# B&R Automation Studio project NAINV104C00R8L515F00 (part 25)

#### Act_Background.st - Change By Project
```iecst
(** 2020-10-08 **)
ACTION Act_Background:

	//Resetting Physical Output
	memset(ADR(a_bPhysicalDO), 0, SIZEOF(a_bPhysicalDO));

	//Digital Output Mapping Physical Output With Config
	IF p_tyDOSettings.diSafetyRlyRst > 0 AND p_tyDOSettings.diSafetyRlyRst <= UDINT_TO_DINT(p_udiMax) THEN
		a_bPhysicalDO[p_tyDOSettings.diSafetyRlyRst]	:= p_bSafetyRlyRst;
	END_IF

	IF p_tyDOSettings.diTLRed > 0 AND p_tyDOSettings.diTLRed <= UDINT_TO_DINT(p_udiMax) THEN
		a_bPhysicalDO[p_tyDOSettings.diTLRed]			:= p_bTLRed;
	END_IF

	IF p_tyDOSettings.diTLAmber > 0 AND p_tyDOSettings.diTLAmber <= UDINT_TO_DINT(p_udiMax) THEN
		a_bPhysicalDO[p_tyDOSettings.diTLAmber]			:= p_bTLAmber;
	END_IF

	IF p_tyDOSettings.diTLGreen > 0 AND p_tyDOSettings.diTLGreen <= UDINT_TO_DINT(p_udiMax) THEN
		a_bPhysicalDO[p_tyDOSettings.diTLGreen]			:= p_bTLGreen;
	END_IF

	IF p_tyDOSettings.diTLWhite > 0 AND p_tyDOSettings.diTLWhite <= UDINT_TO_DINT(p_udiMax) THEN
		a_bPhysicalDO[p_tyDOSettings.diTLWhite]			:= p_bTLWhite;
	END_IF

	IF p_tyDOSettings.diTLBlue > 0 AND p_tyDOSettings.diTLBlue <= UDINT_TO_DINT(p_udiMax) THEN
		a_bPhysicalDO[p_tyDOSettings.diTLBlue]			:= p_bTLBlue;
	END_IF

	IF p_tyDOSettings.diBuz > 0 AND p_tyDOSettings.diBuz <= UDINT_TO_DINT(p_udiMax) THEN
		a_bPhysicalDO[p_tyDOSettings.diBuz]				:= p_bBuz;
	END_IF

	IF p_tyDOSettings.diDBA > 0 AND p_tyDOSettings.diDBA <= UDINT_TO_DINT(p_udiMax) THEN
		a_bPhysicalDO[p_tyDOSettings.diDBA]				:= p_bDBA;
	END_IF

	IF p_tyDOSettings.diDBAStat > 0 AND p_tyDOSettings.diDBAStat <= UDINT_TO_DINT(p_udiMax) THEN
		a_bPhysicalDO[p_tyDOSettings.diDBAStat]			:= p_bDBAStat;
	END_IF

	IF p_tyDOSettings.diUSB > 0 AND p_tyDOSettings.diUSB <= UDINT_TO_DINT(p_udiMax) THEN
		a_bPhysicalDO[p_tyDOSettings.diUSB]				:= p_bUSB;
	END_IF

	IF p_tyDOSettings.diUSB2 > 0 AND p_tyDOSettings.diUSB2 <= UDINT_TO_DINT(p_udiMax) THEN
		a_bPhysicalDO[p_tyDOSettings.diUSB2]			:= p_bUSB2;
	END_IF

	IF p_tyDOSettings.diConvMtrCW > 0 AND p_tyDOSettings.diConvMtrCW <= UDINT_TO_DINT(p_udiMax) THEN
		a_bPhysicalDO[p_tyDOSettings.diConvMtrCW]	:= p_bConvMtrCW;
	END_IF

	IF p_tyDOSettings.diConvMtrCCW > 0 AND p_tyDOSettings.diConvMtrCCW <= UDINT_TO_DINT(p_udiMax) THEN
		a_bPhysicalDO[p_tyDOSettings.diConvMtrCCW]	:= p_bConvMtrCCW;
	END_IF

	IF p_tyDOSettings.diStprUnblkCtrl > 0 AND p_tyDOSettings.diStprUnblkCtrl <= UDINT_TO_DINT(p_udiMax) THEN
		a_bPhysicalDO[p_tyDOSettings.diStprUnblkCtrl]	:= p_bStprUnblkCtrl;
	END_IF

	IF p_tyDOSettings.diStprBlkCtrl > 0 AND p_tyDOSettings.diStprBlkCtrl <= UDINT_TO_DINT(p_udiMax) THEN
		a_bPhysicalDO[p_tyDOSettings.diStprBlkCtrl]		:= p_bStprBlkCtrl;
	END_IF

	IF p_tyDOSettings.diInvertHome > 0 AND p_tyDOSettings.diInvertHome <= UDINT_TO_DINT(p_udiMax) THEN
		a_bPhysicalDO[p_tyDOSettings.diInvertHome]	:= p_bInvertHome;
	END_IF

	IF p_tyDOSettings.diInvertRemote > 0 AND p_tyDOSettings.diInvertRemote <= UDINT_TO_DINT(p_udiMax) THEN
		a_bPhysicalDO[p_tyDOSettings.diInvertRemote]	:= p_bInvertRemote;
	END_IF

	IF p_tyDOSettings.diInvertBrake > 0 AND p_tyDOSettings.diInvertBrake <= UDINT_TO_DINT(p_udiMax) THEN
		a_bPhysicalDO[p_tyDOSettings.diInvertBrake]	:= p_bInvertBrake;
	END_IF

	IF p_tyDOSettings.diClampControl > 0 AND p_tyDOSettings.diClampControl <= UDINT_TO_DINT(p_udiMax) THEN
		a_bPhysicalDO[p_tyDOSettings.diClampControl]	:= p_bClampControl;
	END_IF

	IF p_tyDOSettings.diUnclampControl > 0 AND p_tyDOSettings.diUnclampControl <= UDINT_TO_DINT(p_udiMax) THEN
		a_bPhysicalDO[p_tyDOSettings.diUnclampControl]	:= p_bUnclampControl;
	END_IF

	IF p_tyDOSettings.diMtrPwrRly > 0 AND p_tyDOSettings.diMtrPwrRly <= UDINT_TO_DINT(p_udiMax) THEN
		a_bPhysicalDO[p_tyDOSettings.diMtrPwrRly]	:= p_bMtrPwrRly;
	END_IF

	IF p_tyDOSettings.diInShutterOpenCtrl > 0 AND p_tyDOSettings.diInShutterOpenCtrl <= UDINT_TO_DINT(p_udiMax) THEN
		a_bPhysicalDO[p_tyDOSettings.diInShutterOpenCtrl]	:= p_bInShutterOpenCtrl;
	END_IF

	IF p_tyDOSettings.diInShutterCloseCtrl > 0 AND p_tyDOSettings.diInShutterCloseCtrl <= UDINT_TO_DINT(p_udiMax) THEN
		a_bPhysicalDO[p_tyDOSettings.diInShutterCloseCtrl]	:= p_bInShutterCloseCtrl;
	END_IF

	IF p_tyDOSettings.diOutShutterOpenCtrl > 0 AND p_tyDOSettings.diOutShutterOpenCtrl <= UDINT_TO_DINT(p_udiMax) THEN
		a_bPhysicalDO[p_tyDOSettings.diOutShutterOpenCtrl]	:= p_bOutShutterOpenCtrl;
	END_IF

	IF p_tyDOSettings.diOutShutterCloseCtrl > 0 AND p_tyDOSettings.diOutShutterCloseCtrl <= UDINT_TO_DINT(p_udiMax) THEN
		a_bPhysicalDO[p_tyDOSettings.diOutShutterCloseCtrl]	:= p_bOutShutterCloseCtrl;
	END_IF

	IF p_tyDOSettings.diClamp1Ctrl > 0 AND p_tyDOSettings.diClamp1Ctrl <= UDINT_TO_DINT(p_udiMax) THEN
		a_bPhysicalDO[p_tyDOSettings.diClamp1Ctrl]	:= p_bClamp1Ctrl;
	END_IF

	IF p_tyDOSettings.diUnClamp1Ctrl > 0 AND p_tyDOSettings.diUnClamp1Ctrl <= UDINT_TO_DINT(p_udiMax) THEN
		a_bPhysicalDO[p_tyDOSettings.diUnClamp1Ctrl]	:= p_bUnClamp1Ctrl;
	END_IF

	IF p_tyDOSettings.diClamp2Ctrl > 0 AND p_tyDOSettings.diClamp2Ctrl <= UDINT_TO_DINT(p_udiMax) THEN
		a_bPhysicalDO[p_tyDOSettings.diClamp2Ctrl]	:= p_bClamp2Ctrl;
	END_IF

	IF p_tyDOSettings.diUnClamp2Ctrl > 0 AND p_tyDOSettings.diUnClamp2Ctrl <= UDINT_TO_DINT(p_udiMax) THEN
		a_bPhysicalDO[p_tyDOSettings.diUnClamp2Ctrl]	:= p_bUnClamp2Ctrl;
	END_IF

	IF p_tyDOSettings.diClamp3Ctrl > 0 AND p_tyDOSettings.diClamp3Ctrl <= UDINT_TO_DINT(p_udiMax) THEN
		a_bPhysicalDO[p_tyDOSettings.diClamp3Ctrl]	:= p_bClamp3Ctrl; //
	END_IF

	IF p_tyDOSettings.diUnClamp3Ctrl > 0 AND p_tyDOSettings.diUnClamp3Ctrl <= UDINT_TO_DINT(p_udiMax) THEN
		a_bPhysicalDO[p_tyDOSettings.diUnClamp3Ctrl]	:= p_bUnClamp3Ctrl;
	END_IF

	// ADD
	IF p_bHermesUSCmdFeaturePause THEN
		IF p_tyHermesUSCmdPause.bFeatureRequestFrom  THEN
			//a_bPhysicalDO[p_tyDOSettings.diMachineSafetySigToUS]	:= p_tyHermesUSCmdPause.bMachineSafetySigTo;
			p_tyHermesUSCmdPause.bMachineSafetySigTo				:= p_bMachineSafetySigToUS;
		END_IF
		IF p_tyHermesUSCmdPause.bFeatureRequestTo THEN
			//a_bPhysicalDO[p_tyDOSettings.diTopCvrUnlckToUS]	:= p_tyHermesUSCmdPause.bUnlockCoverSigTo;
			p_tyHermesUSCmdPause.bUnlockCoverSigTo					:= p_bTopCvrUnlckToUS;
		END_IF
	ELSE
		IF p_tyDOSettings.diMachineSafetySigToUS > 0 AND p_tyDOSettings.diMachineSafetySigToUS  <= UDINT_TO_DINT(p_udiMax) THEN
			a_bPhysicalDO[p_tyDOSettings.diMachineSafetySigToUS]	:= p_bMachineSafetySigToUS;
		END_IF
		IF p_tyDOSettings.diTopCvrUnlckToUS > 0 AND p_tyDOSettings.diTopCvrUnlckToUS  <= UDINT_TO_DINT(p_udiMax) THEN
			a_bPhysicalDO[p_tyDOSettings.diTopCvrUnlckToUS]	:= p_bTopCvrUnlckToUS;
		END_IF
	END_IF
	IF p_bHermesDSCmdFeaturePause THEN
		IF p_tyHermesDSCmdPause.bFeatureRequestTo THEN
			//a_bPhysicalDO[p_tyDOSettings.diMachineSafetySigToDS]	:= p_tyHermesDSCmdPause.bMachineSafetySigTo;
			p_tyHermesDSCmdPause.bMachineSafetySigTo  				:= p_bMachineSafetySigToDS;
		END_IF
		IF p_tyHermesDSCmdPause.bFeatureRequestFrom THEN
			//a_bPhysicalDO[p_tyDOSettings.diTopCvrUnlckToDS]	:= p_tyHermesDSCmdPause.bUnlockCoverSigTo;
			p_tyHermesDSCmdPause.bUnlockCoverSigTo					:= p_bTopCvrUnlckToDS;
		END_IF
	ELSE
		IF p_tyDOSettings.diMachineSafetySigToDS  > 0 AND p_tyDOSettings.diMachineSafetySigToDS  <= UDINT_TO_DINT(p_udiMax) THEN
			a_bPhysicalDO[p_tyDOSettings.diMachineSafetySigToDS]	:= p_bMachineSafetySigToDS;
		END_IF
		IF p_tyDOSettings.diTopCvrUnlckToDS > 0 AND p_tyDOSettings.diTopCvrUnlckToDS  <= UDINT_TO_DINT(p_udiMax) THEN
			a_bPhysicalDO[p_tyDOSettings.diTopCvrUnlckToDS]	:= p_bTopCvrUnlckToDS;
		END_IF
	END_IF

	IF p_tyDOSettings.diSafetyTopCoverSWCoil1  > 0 AND p_tyDOSettings.diSafetyTopCoverSWCoil1  <= UDINT_TO_DINT(p_udiMax) THEN
		a_bPhysicalDO[p_tyDOSettings.diSafetyTopCoverSWCoil1]	:= p_bSafetyTopCoverSWCoil1;
	END_IF
	IF p_tyDOSettings.diCoverPBLED1 > 0 AND p_tyDOSettings.diCoverPBLED1  <= UDINT_TO_DINT(p_udiMax) THEN
		a_bPhysicalDO[p_tyDOSettings.diCoverPBLED1]	:= p_bCoverPBLED1;
	END_IF
	IF p_tyDOSettings.diBypassTopCover1 > 0 AND p_tyDOSettings.diBypassTopCover1  <= UDINT_TO_DINT(p_udiMax) THEN
		a_bPhysicalDO[p_tyDOSettings.diBypassTopCover1]	:= p_bBypsCoverSW1;
	END_IF

	//Update Output
	tyDOutput.bSafetyRlyRst			:= p_bSafetyRlyRst;
	tyDOutput.bTLWhite				:= p_bTLWhite;
	tyDOutput.bTLAmber				:= p_bTLAmber;
	tyDOutput.bTLGreen				:= p_bTLGreen;
	tyDOutput.bTLRed				:= p_bTLRed;
	tyDOutput.bTLBlue				:= p_bTLBlue;
	tyDOutput.bBuz					:= p_bBuz;
	tyDOutput.bUSB					:= p_bUSB;
	tyDOutput.bDBA					:= p_bDBA;
	tyDOutput.bDBAStat				:= p_bDBAStat;
	tyDOutput.bUSB2					:= p_bUSB2; //ADD_2023_0032B01
	tyDOutput.bConvMtrCW			:= p_bConvMtrCW;
	tyDOutput.bConvMtrCCW			:= p_bConvMtrCCW;
	tyDOutput.bStprUnblkCtrl		:= p_bStprUnblkCtrl;
	tyDOutput.bStprBlkCtrl			:= p_bStprBlkCtrl;
	tyDOutput.bInvertHome			:= p_bInvertHome;
	tyDOutput.bInvertRemote			:= p_bInvertRemote;
	tyDOutput.bInvertBrake			:= p_bInvertBrake;
	tyDOutput.bClampControl			:= p_bClampControl;
	tyDOutput.bUnclampControl		:= p_bUnclampControl;
	tyDOutput.bMtrPwrRly			:= p_bMtrPwrRly;
	tyDOutput.bInShutterOpenCtrl	:= p_bInShutterOpenCtrl;
	tyDOutput.bInShutterCloseCtrl	:= p_bInShutterCloseCtrl;
	tyDOutput.bOutShutterOpenCtrl	:= p_bOutShutterOpenCtrl;
	tyDOutput.bOutShutterCloseCtrl	:= p_bOutShutterCloseCtrl;
	tyDOutput.bClamp1Ctrl			:= p_bClamp1Ctrl;
	tyDOutput.bUnClamp1Ctrl			:= p_bUnClamp1Ctrl;
	tyDOutput.bClamp2Ctrl			:= p_bClamp2Ctrl;
	tyDOutput.bUnClamp2Ctrl			:= p_bUnClamp2Ctrl;
	tyDOutput.bClamp3Ctrl			:= p_bClamp3Ctrl;
	tyDOutput.bUnClamp3Ctrl			:= p_bUnClamp3Ctrl;

	// ADD
	tyDOutput.bMachineSafetySigToDS :=p_bMachineSafetySigToDS;
	tyDOutput.bMachineSafetySigToUS := p_bMachineSafetySigToUS;
	tyDOutput.bSafetyTopCoverSWCoil1 := p_bSafetyTopCoverSWCoil1;
	tyDOutput.bBypassTopCover1 := p_bBypsCoverSW1;
	tyDOutput.bCoverPBLED1 := p_bCoverPBLED1;
	tyDOutput.bTopCvrUnlckToDS := p_bMachineSafetySigToUS;
	tyDOutput.bTopCvrUnlckToUS := p_bMachineSafetySigToDS;
END_ACTION
```

#### InputRef.var - Change By Project
```iecst
(*2020-10-08*)
(**)
(*General*)
VAR
	p_eAct : REFERENCE TO eDOAction;
	p_udiMax : REFERENCE TO UDINT;
END_VAR
(**)
(*Configuration*)
VAR
	p_tyDOSettings : REFERENCE TO tyDigitalOutputSettings;
END_VAR
(**)
VAR
	p_bManual : REFERENCE TO BOOL;
	p_bSafetyRlyRst : REFERENCE TO BOOL;
	p_bTLRed : REFERENCE TO BOOL;
	p_bTLAmber : REFERENCE TO BOOL;
	p_bTLGreen : REFERENCE TO BOOL;
	p_bTLWhite : REFERENCE TO BOOL;
	p_bTLBlue : REFERENCE TO BOOL;
	p_bBuz : REFERENCE TO BOOL;
	p_bUSB : REFERENCE TO BOOL;
	p_bDBA : REFERENCE TO BOOL;
	p_bDBAStat : REFERENCE TO BOOL;
	p_bUSB2 : REFERENCE TO BOOL;
	p_bConvMtrCW : REFERENCE TO BOOL;
	p_bConvMtrCCW : REFERENCE TO BOOL;
	p_bStprUnblkCtrl : REFERENCE TO BOOL;
	p_bStprBlkCtrl : REFERENCE TO BOOL;
	p_bInvertBrake : REFERENCE TO BOOL;
	p_bInvertHome : REFERENCE TO BOOL;
	p_bInvertRemote : REFERENCE TO BOOL;
	p_bClampControl : REFERENCE TO BOOL;
	p_bUnclampControl : REFERENCE TO BOOL;
	p_bMtrPwrRly : REFERENCE TO BOOL;
	p_bInShutterOpenCtrl : REFERENCE TO BOOL;
	p_bInShutterCloseCtrl : REFERENCE TO BOOL;
	p_bOutShutterOpenCtrl : REFERENCE TO BOOL;
	p_bOutShutterCloseCtrl : REFERENCE TO BOOL;
	p_bClamp1Ctrl : REFERENCE TO BOOL;
	p_bUnClamp1Ctrl : REFERENCE TO BOOL;
	p_bClamp2Ctrl : REFERENCE TO BOOL;
	p_bUnClamp2Ctrl : REFERENCE TO BOOL;
	p_bClamp3Ctrl : REFERENCE TO BOOL;
	p_bUnClamp3Ctrl : REFERENCE TO BOOL;
END_VAR
(**)
VAR
	p_bLinkConvMtrSigOnOrLToR : REFERENCE TO BOOL;
	p_bLinkConvMtrDirOrRToL : REFERENCE TO BOOL;
	p_eLinkOpsInvertInvertCurrPos : REFERENCE TO eInvertPos;
	p_bLinkUIConvDCCtrl : REFERENCE TO BOOL;
	p_bLinkUIInvertDCCtrl : REFERENCE TO BOOL;
	p_usiLinkProdRcpCurrRcpMcMod : REFERENCE TO USINT;
	p_eConvStatus : REFERENCE TO eFBStatus;
	p_bLinkOpsInvertStepInitTwdStpr : REFERENCE TO BOOL;
	p_bLinkOpsInvertStepInitAwayStpr : REFERENCE TO BOOL;
END_VAR
(**)
VAR
	p_tyDI : REFERENCE TO tyDigitalInput;
END_VAR
(**)
VAR
	p_bBypsCoverSW1 : REFERENCE TO BOOL;
	p_bTopCvrUnlckToDS : REFERENCE TO BOOL;
	p_bTopCvrUnlckToUS : REFERENCE TO BOOL;
	p_bMachineSafetySigToDS : REFERENCE TO BOOL;
	p_bMachineSafetySigToUS : REFERENCE TO BOOL;
	p_bSafetyTopCoverSWCoil1 : REFERENCE TO BOOL;
	p_bCoverPBLED1 : REFERENCE TO BOOL;
END_VAR
(**)
VAR
	p_bHermesCmdInitialCompl : REFERENCE TO BOOL;
	p_bHermesUSCmdFeaturePause : REFERENCE TO BOOL;
	p_tyHermesUSCmdPause : REFERENCE TO tyHermesCommandPause;
	p_bHermesDSCmdFeaturePause : REFERENCE TO BOOL;
	p_tyHermesDSCmdPause : REFERENCE TO tyHermesCommandPause;
END_VAR
```

#### Local.var - Change By Project
```iecst
(*2020-10-08*)
(**)
(*Local Action, State & Status*)
VAR
	eAct : eDOAction := DOActIdle;
	eStat : eDOAction := DOActIdle;
	eStatus : eFBStatus := Idle;
	sStatTxt : STRING[200] := '';
	a_sStatText : ARRAY[0..50] OF STRING[200] := ['Idling','Resetting All Special Output','Turning On Bypass Cover Switch','Turning Off Bypass Cover Switch',47('')];
END_VAR
(**)
(*Local Alarm*)
(**)
(*Local Output*)
VAR
	tyDOutput : tyDigitalOutput;
END_VAR
(**)
(*Local Input*)
VAR
	tyDOSettings : tyDigitalOutputSettings;
END_VAR
(**)
VAR
	bManual : BOOL := FALSE;
	bSafetyRlyRst : BOOL := FALSE;
	bTLRed : BOOL := FALSE;
	bTLAmber : BOOL := FALSE;
	bTLGreen : BOOL := FALSE;
	bTLBlue : BOOL := FALSE;
	bTLWhite : BOOL := FALSE;
	bBuz : BOOL := FALSE;
	bUSB : BOOL := FALSE;
	bDBA : BOOL := FALSE;
	bDBAStat : BOOL := FALSE;
	bUSB2 : BOOL := FALSE;
	bConvMtrCW : BOOL := FALSE;
	bConvMtrCCW : BOOL := FALSE;
	bStprUnblkCtrl : BOOL := FALSE;
	bStprBlkCtrl : BOOL := FALSE;
	bInvertHome : BOOL := FALSE;
	bInvertRemote : BOOL := FALSE;
	bInvertBrake : BOOL := FALSE;
	bClampControl : BOOL := FALSE;
	bUnclampControl : BOOL := FALSE;
	bMtrPwrRly : BOOL := TRUE;
	bInShutterOpenCtrl : BOOL;
	bInShutterCloseCtrl : BOOL;
	bOutShutterOpenCtrl : BOOL;
	bOutShutterCloseCtrl : BOOL;
	bClamp1Ctrl : BOOL;
	bUnClamp1Ctrl : BOOL;
	bClamp2Ctrl : BOOL;
	bUnClamp2Ctrl : BOOL;
	bClamp3Ctrl : BOOL;
	bUnClamp3Ctrl : BOOL;
	bBypassTopCover1 : BOOL;
	bTopCvrUnlckToDS : BOOL;
	bTopCvrUnlckToUS : BOOL;
	bMachineSafetySigToDS : BOOL;
	bMachineSafetySigToUS : BOOL;
	bCoverPBLED1 : BOOL;
	bSafetyTopCoverSWCoil1 : BOOL;
END_VAR
(**)
(*Local*)
VAR
	bInitDone : BOOL;
	bInitialDone : BOOL;
	a_bPhysicalDO : ARRAY[1..c_udiDOutputMax] OF BOOL;
	eStatOld : eDOAction := DOActIdle;
	bHermesDummyMem : BOOL;
END_VAR
```

### Hermes.typ - Do Not Change!!!
```iecst
(*2019-05-04*)
(**)
(*Action*)

TYPE
	eHermesAction :
		(
		HermesActIdle,
		HermesActBGStartRun,
		HermesActBGStopRun,
		HermesActDeleteOldLog,
		HermesActCreateDir,
		HermesActWriteRetain,
		HermesActWriteRetainLane1,
		HermesActWriteRetainLane2,
		HermesActWriteRetainLane3,
		HermesActWriteRetainLane4,
		HermesActReadRetain,
		HermesActReadRetainLane1,
		HermesActReadRetainLane2,
		HermesActReadRetainLane3,
		HermesActReadRetainLane4,
		HermesActWriteConfig,
		HermesActReadConfig
		);
END_TYPE

(**)

TYPE
	tyHermesConfiguration : 	STRUCT
		a_tyUSParam : ARRAY[0..c_diHermesConfigMaxIdx]OF tyHermesUSParam;
		a_tyDSParam : ARRAY[0..c_diHermesConfigMaxIdx]OF tyHermesDSParam;
		tySvyParam : tyHermesSvyParam;
	END_STRUCT;
	tyHermesDSParam : 	STRUCT
		tSndAlive : TIME;
		tRcvAlive : TIME;
		sDownstreamInterfaceId : STRING[80]; (*The ID of the transportation interface on the downstream side*)
		uiSvrPort : UINT;
		iLaneID : INT;
		sMachineId : STRING[80] := '';
		sClientAddress : STRING[15] := '';
		uiClientPort : UINT;
		bFeatureCheckAliveResponse : BOOL;
		bFeatureBoardForecast : BOOL;
		bFeatureSendBoardInfo : BOOL;
		bFeatureCommand : BOOL;
	END_STRUCT;
	tyHermesUSParam : 	STRUCT
		tSndAlive : TIME;
		tRcvAlive : TIME;
		uiClntPort : UINT;
		iLaneID : INT;
		sMachineId : STRING[80] := '';
		sHostAddress : STRING[15] := '';
		uiHostPort : UINT;
		sUpstreamInterfaceId : STRING[80]; (*The ID of the transportation interface on the upstream side*)
		bFeatureCheckAliveResponse : BOOL;
		bFeatureBoardForecast : BOOL;
		bFeatureQueryBoardInfo : BOOL;
		bFeatureCommand : BOOL;
		bCmpTypeId : BOOL;
		bCmpParam : BOOL;
		bOverwrite : BOOL;
	END_STRUCT;
	tyHermesRmtParam : 	STRUCT
		uiSvrPort : UINT;
	END_STRUCT;
	tyHermesSvyParam : 	STRUCT
		tSndAlive : TIME;
		tRcvAlive : TIME;
		uiSvySvstemPort : UINT;
		iLaneID : INT;
		sMachineId : STRING[80];
		sClientAddress : STRING[15];
		uiClientPort : UINT;
		bFeatureCheckAliveResponse : BOOL;
		bFeatureConfiguration : BOOL;
		bFeatureBoardTracking : BOOL;
		bFeatureQueryWorkOrderInfo : BOOL;
		bFeatureSendWorkOrderInfo : BOOL;
		bFeatureInsertBrd : BOOL;
	END_STRUCT;
	tyHermesBrdAvlDat : 	STRUCT
		a_tyXMLTableDataBrdAvl : ARRAY[0..200]OF tyXMLTableDat;
		iXMLTableDataBrdAvlTtlIdx : INT;
		bNewBrdAvl : BOOL := TRUE;
	END_STRUCT;
END_TYPE
```

### Hermes.var - Change By Project
```iecst
(*2019-05-04*)
(**)
(*Action & State & Status*)
VAR
	p_HermesStat : UDINT;
	p_HermesStatus : UDINT;
	p_HermesStatTxt : UDINT;
END_VAR
(**)
(*Alarm*)
VAR
	p_HermesAlmData : UDINT;
END_VAR
(**)
(*Output*)
VAR
	p_HermesFileNotFound : UDINT;
	p_HermesConfiguration : UDINT;
	p_HermesConfigurationWr : UDINT;
	p_HermesUSParam1 : UDINT;
	p_HermesUSParam2 : UDINT;
	p_HermesUSParam3 : UDINT;
	p_HermesDSParam1 : UDINT;
	p_HermesDSParam2 : UDINT;
	p_HermesDSParam3 : UDINT;
	p_HermesSvyParam : UDINT;
	p_HermesBrdAvlDataTable1stZ : UDINT;
	p_HermesBrdAvlDataTtlIdx1stZ : UDINT;
	p_HermesBrdAvlDataNewBrdAvl1stZ : UDINT;
	p_HermesBrdAvlDataTableLastZ : UDINT;
	p_HermesBrdAvlDataTtlIdxLastZ : UDINT;
	p_HermesBrdAvlDataNewBrdAvlLastZ : UDINT;
	pa_HermesDSParam : UDINT;
	p_HermesReverseDS1SendBFId : UDINT;
	p_HermesReverseDS2SendBFId : UDINT;
	p_HermesSwitchtoReverseTransport : UDINT;
	p_HermesEntToReversePosition : UDINT;
	p_HermesCmdInitialCompl : UDINT;
	p_HermesUSCmdFeaturePause : UDINT;
	p_HermesUSCmdPause : UDINT;
	p_HermesDSCmdFeaturePause : UDINT;
	p_HermesDSCmdPause : UDINT;
END_VAR
```

### Program Logical/Hermes/Hermes (IEC, version 1.00.0) - 1.00.0 - NtHermes v5.00.0 , NtTCP v5.00.0 , NtMessage v5.00.0

#### Init.st - Change By Project
```iecst
(** 2019-05-04 **)
PROGRAM _INIT

	(* Always Change If Project Change *)

	//Pass Address To Global Address For External Use
	//Action, State & Status
	p_HermesStat	:= ADR(eStat);
	p_HermesStatus	:= ADR(eStatus);
	p_HermesStatTxt	:= ADR(sStatTxt);

	//Alarm
	p_HermesAlmData	:= ADR(tyAlmData);

	//Output
	p_HermesFileNotFound		:= ADR(bFileNotFound);
	p_HermesConfiguration		:= ADR(tyCurrConfiguration);
	p_HermesConfigurationWr	    := ADR(tyConfigurationWr);
	p_HermesUSParam1			:= ADR(tyCurrConfiguration.a_tyUSParam[0]);
	p_HermesUSParam2			:= ADR(tyCurrConfiguration.a_tyUSParam[1]);
	p_HermesUSParam3			:= ADR(tyCurrConfiguration.a_tyUSParam[2]);
	p_HermesDSParam1			:= ADR(tyCurrConfiguration.a_tyDSParam[0]);
	p_HermesDSParam2			:= ADR(tyCurrConfiguration.a_tyDSParam[1]);
	p_HermesDSParam3			:= ADR(tyCurrConfiguration.a_tyDSParam[2]);
	p_HermesSvyParam		    := ADR(tyCurrConfiguration.tySvyParam);
	p_HermesBrdAvlDataTable1stZ		    := ADR(a_tyHermesBrdAvlData[1].a_tyXMLTableDataBrdAvl); //Lane 1 First Zone Data, for B.F
	p_HermesBrdAvlDataTtlIdx1stZ    	:= ADR(a_tyHermesBrdAvlData[1].iXMLTableDataBrdAvlTtlIdx);  //Lane 1 First Zone Data, for B.F
	p_HermesBrdAvlDataNewBrdAvl1stZ	    := ADR(a_tyHermesBrdAvlData[1].bNewBrdAvl);  //Lane 1 First Zone Data, for B.F
	p_HermesBrdAvlDataTableLastZ		:= ADR(a_tyHermesBrdAvlData[1].a_tyXMLTableDataBrdAvl); //Lane 1 Last Zone Data,for B.A, adjust array no. accordingly
	p_HermesBrdAvlDataTtlIdxLastZ	    := ADR(a_tyHermesBrdAvlData[1].iXMLTableDataBrdAvlTtlIdx); //Lane 1 Last Zone Data,for B.A, adjust array no. accordingly
	p_HermesBrdAvlDataNewBrdAvlLastZ	:= ADR(a_tyHermesBrdAvlData[1].bNewBrdAvl); //Lane 1 Last Zone Data,for B.A, adjust array no. accordingly
	(* Always Change If Project Change *)
	p_HermesCmdInitialCompl		:= ADR(bCmdInitialCompl);

	//check route
	pa_HermesDSParam			:= ADR(tyCurrConfiguration.a_tyDSParam);

	//route output signal
	p_HermesReverseDS1SendBFId	:= ADR(usiReverseDS1SndBfWBrdID);
	p_HermesReverseDS2SendBFId	:= ADR(usiReverseDS2SndBfWBrdID);

	p_HermesSwitchtoReverseTransport := ADR(bSwitchtoReverseTransport);
	p_HermesEntToReversePosition := ADR(bEntToReversePosition);
	//p_HermesBrdAvlDataNewBrdAvlLastZ
END_PROGRAM
```

#### Act_InitGlobal.st - Change By Project
```iecst
(** 2019-05-04 **)
ACTION Act_InitGlobal:

	(* Always Change If Project Change *)

	//Pass Data To Link
	p_bLinkStartupRun ACCESS p_StartupRun;

	p_eLinkMcParamUSCommMod ACCESS p_McParamUSCommMod;
	p_eLinkMcParamUSComm2Mod ACCESS p_McParamUSComm2Mod;

	p_bLinkOpsInvertStepInitDone ACCESS p_OpsInvertStepInitDone;
	p_bLinkOpsInvertStepEntToEnd ACCESS p_OpsInvertStepEntToEnd;
	p_bLinkOpsInvertStepEntToInOff ACCESS p_OpsInvertStepEntToInOff;
	p_bLinkOpsInvertStepExitBrd ACCESS p_OpsInvertStepExitBrd;
	p_bLinkConvHvBrd ACCESS p_ConvHvBrd;//p_OpsInvertHvBrd;
	p_bLinkOpsInvertStepInvert ACCESS p_OpsInvertStepInvert;

	//p_tyUSHermestyBoardAvailable ACCESS p_USHermestyBoardAvailable;
	//Pass Data To Internal Use

	p_eAct ACCESS ADR(eAct);
	p_udiRstErr ACCESS p_RstErrReset;
	p_bPrep ACCESS p_NtParamHermesPrep;
	pa_tyUSParam ACCESS p_UIHermesUSParamWr;
	pa_tyDSParam ACCESS p_UIHermesDSParamWr;
	p_tySvyParam ACCESS p_UIHermesSvyParamWr; //HMI Svy Configure from UI
	p_tyRmtSetConfiguration ACCESS p_RmtHermesSetConfiguration; //US,DS SetConfigure from RmtHermes
	p_tySvySetConfiguration ACCESS p_SvyHermesSetConfiguration; //US,DS SetConfigure from SvyHermes

	//p_tySvySetConfiguration ACCESS p_SvyHermesSetConfiguration; //US,DS SetConfigure from SvyHermes
	p_bRmtPrep ACCESS p_NtParamHermesRmtPrep;
	p_bRmtEn ACCESS p_McParamHermesRmtEn;
	p_bSvyPrep ACCESS ADR(bSvyPrep);
	p_bSvyEn ACCESS ADR(bSvyEn);
	p_sRetainFileName1 ACCESS ADR(sRetainFileName1);
	p_sRetainFileName2 ACCESS ADR(sRetainFileName2);
	p_sRetainFileName3 ACCESS ADR(sRetainFileName3);
	p_sRetainFileName4 ACCESS ADR(sRetainFileName4);
	p_udiRetainDataAddr1 ACCESS ADR(udiRetainDataAddr1);
	p_udiRetainDataLen1 ACCESS ADR(udiRetainDataLen1);
	p_udiRetainDataAddr2 ACCESS ADR(udiRetainDataAddr2);
	p_udiRetainDataLen2 ACCESS ADR(udiRetainDataLen2);
	p_udiRetainDataAddr3 ACCESS ADR(udiRetainDataAddr3);
	p_udiRetainDataLen3 ACCESS ADR(udiRetainDataLen3);
	p_udiRetainDataAddr4 ACCESS ADR(udiRetainDataAddr4);
	p_udiRetainDataLen4 ACCESS ADR(udiRetainDataLen4);

	p_sConfigFileName ACCESS p_NtParamHermesConfigFileNm;
	p_sProgNm ACCESS p_NtParamHermesProgNm;
	p_bNtSettingsLoadDone ACCESS p_StartupNtSettingsLoadDone;
	p_bRmtHermesWriteConfig ACCESS p_RmtHermesWriteConfig;
	//p_bSvyHermesWriteConfig ACCESS p_SvyHermesWriteConfig;
	p_bUISaveHMIConfigure ACCESS p_UISaveHMIConfigure;
	p_bUISaveHMISvyConfig ACCESS p_UISaveHMISvyConfig;
	p_sMcId ACCESS p_McParamMcNm;

	p_bRmtFoundIndexUS1 ACCESS p_RmtHermesFoundIndexUS1;
	p_bRmtFoundIndexUS2 ACCESS p_RmtHermesFoundIndexUS2;
	p_bRmtFoundIndexUS3 ACCESS p_RmtHermesFoundIndexUS3;
	p_bRmtFoundIndexUS4 ACCESS p_RmtHermesFoundIndexUS4;
	p_bRmtFoundIndexDS1 ACCESS p_RmtHermesFoundIndexDS1;
	p_bRmtFoundIndexDS2 ACCESS p_RmtHermesFoundIndexDS2;
	p_bRmtFoundIndexDS3 ACCESS p_RmtHermesFoundIndexDS3;
	p_bRmtFoundIndexDS4 ACCESS p_RmtHermesFoundIndexDS4;
	p_udiRmtIndexUS1 ACCESS p_RmtHermesIndexUS1;
	p_udiRmtIndexUS2 ACCESS p_RmtHermesIndexUS2;
	p_udiRmtIndexUS3 ACCESS p_RmtHermesIndexUS3;
	p_udiRmtIndexUS4 ACCESS p_RmtHermesIndexUS4;
	p_udiRmtIndexDS1 ACCESS p_RmtHermesIndexDS1;
	p_udiRmtIndexDS2 ACCESS p_RmtHermesIndexDS2;
	p_udiRmtIndexDS3 ACCESS p_RmtHermesIndexDS3;
	p_udiRmtIndexDS4 ACCESS p_RmtHermesIndexDS4;

	p_bSvyFoundIndexUS1 ACCESS p_SvyHermesFoundIndexUS1;
	p_bSvyFoundIndexUS2 ACCESS p_SvyHermesFoundIndexUS2;
	p_bSvyFoundIndexUS3 ACCESS p_SvyHermesFoundIndexUS3;
	p_bSvyFoundIndexUS4 ACCESS p_SvyHermesFoundIndexUS4;
	p_bSvyFoundIndexDS1 ACCESS p_SvyHermesFoundIndexDS1;
	p_bSvyFoundIndexDS2 ACCESS p_SvyHermesFoundIndexDS2;
	p_bSvyFoundIndexDS3 ACCESS p_SvyHermesFoundIndexDS3;
	p_bSvyFoundIndexDS4 ACCESS p_SvyHermesFoundIndexDS4;
	p_udiSvyIndexUS1 ACCESS p_SvyHermesIndexUS1;
	p_udiSvyIndexUS2 ACCESS p_SvyHermesIndexUS2;
	p_udiSvyIndexUS3 ACCESS p_SvyHermesIndexUS3;
	p_udiSvyIndexUS4 ACCESS p_SvyHermesIndexUS4;
	p_udiSvyIndexDS1 ACCESS p_SvyHermesIndexDS1;
	p_udiSvyIndexDS2 ACCESS p_SvyHermesIndexDS2;
	p_udiSvyIndexDS3 ACCESS p_SvyHermesIndexDS3;
	p_udiSvyIndexDS4 ACCESS p_SvyHermesIndexDS4;

	//Command
	//Unlock Cover
	p_bNTParamUnlockCovPrep ACCESS p_NTParamUnlockCovPrep;
	p_bNTParamMachineSafetySig ACCESS p_NTParamMachineSafetySig;

	//route
	p_bOpsInvertStepInitDone ACCESS p_OpsInvertStepInitDone;
	p_bOpsInvertHvBrd ACCESS p_OpsInvertHvBrd;
	(* Always Change If Project Change *)

END_ACTION
```

#### InputRef_Link.var - Change By Project
```iecst
(*2019-05-04*)
(**)
VAR
	p_bLinkStartupRun : REFERENCE TO BOOL;
END_VAR
(**)
VAR
	p_eLinkMcParamUSCommMod : REFERENCE TO eMcSetCommMod;
	p_eLinkMcParamUSComm2Mod : REFERENCE TO eMcSetCommMod;
	pa_tyLinkXMLTableDataBrdAvl : REFERENCE TO ARRAY[0..200] OF tyXMLTableDat;
	p_iLinkXMLTableDataBrdAvlTtlIdx : REFERENCE TO INT;
END_VAR
(**)
VAR
	p_bLinkOpsInvertStepInitDone : REFERENCE TO BOOL;
	p_bLinkOpsInvertStepEntToEnd : REFERENCE TO BOOL;
	p_bLinkOpsInvertStepEntToInOff : REFERENCE TO BOOL;
	p_bLinkOpsInvertStepExitBrd : REFERENCE TO BOOL;
	p_bLinkConvHvBrd : REFERENCE TO BOOL;
	p_bLinkOpsInvertStepInvert : REFERENCE TO BOOL;
	p_tyUSHermestyBoardAvailable : REFERENCE TO tyHermesBoardAvailable;
END_VAR
(**)
VAR
	tyHermesBrdAvlData : tyHermesBrdAvlDat;
	a_tyHermesBrdAvlData : ARRAY[0..6] OF tyHermesBrdAvlDat; (*Cater Up to 6 Zones*)
	bHermesWriteRetain : BOOL;
	sLowerCase : STRING[254] := '';
END_VAR
```

#### Act_LinkAction.st - Change By Project
```iecst
(** 2019-05-04 **)
ACTION Act_LinkAction:

	IF p_bLinkStartupRun = TRUE THEN
		p_eAct ACCESS p_StartupHermesAct;
//	ELSIF p_bSvyHermesWriteConfig THEN
//		p_eAct ACCESS p_SvyHermesAct;
	ELSIF p_bRmtHermesWriteConfig THEN
		p_eAct ACCESS p_RmtHermesAct;
	ELSIF p_bUISaveHMIConfigure OR p_bUISaveHMISvyConfig THEN
		p_eAct ACCESS p_UIHermesAct;
	END_IF

END_ACTION
```

#### Act_LinkEn.st - Change By Project
```iecst
(** 2019-05-04 **)
ACTION Act_LinkEn:

	//Link bPrep, bEn & bDis

END_ACTION
```

#### Act_Link.st - Change By Project
```iecst
(** 2019-05-04 **)
ACTION Act_Link:

	IF p_bLinkStartupRun = FALSE THEN

		//Passing Board Available Memory
		//Init Board
		IF EDGEPOS(p_bLinkOpsInvertStepInitDone = TRUE) THEN

			IF p_bLinkConvHvBrd = FALSE THEN
				//tyHermesBrdAvlData.bNewBrdAvl	:= TRUE;
				a_tyHermesBrdAvlData[1].bNewBrdAvl := TRUE;
				bHermesWriteRetainLane1	:= TRUE;
			END_IF

		END_IF

		//Enter Board - US1
		IF EDGEPOS(p_bLinkConvHvBrd) AND (p_bLinkOpsInvertStepEntToEnd = TRUE OR p_bLinkOpsInvertStepEntToInOff) THEN

			IF p_eLinkMcParamUSCommMod = McSetCommModHermes THEN

				a_tyHermesBrdAvlData[1].a_tyXMLTableDataBrdAvl		:= pa_tyLinkXMLTableDataBrdAvl;
				a_tyHermesBrdAvlData[1].iXMLTableDataBrdAvlTtlIdx	:= p_iLinkXMLTableDataBrdAvlTtlIdx;
				a_tyHermesBrdAvlData[1].bNewBrdAvl					:= FALSE;

				bHermesWriteRetainLane1	:= TRUE;

			ELSE

				a_tyHermesBrdAvlData[1].bNewBrdAvl	:= TRUE;

				bHermesWriteRetainLane1	:= TRUE;

			END_IF

		END_IF

		//Exit Board
		IF p_bLinkOpsInvertStepExitBrd = TRUE AND EDGENEG(p_bLinkConvHvBrd) THEN
			a_tyHermesBrdAvlData[1].bNewBrdAvl	:= TRUE;

			bHermesWriteRetainLane1	:= TRUE;
		END_IF

		//Write Hermes Retain Data
		IF bHermesWriteRetainLane1 = TRUE AND eStatus <> Busy THEN
			p_eAct	:= HermesActWriteRetain;

			IF (eStat = HermesActWriteRetain) AND (eStatus = Done) THEN
				p_eAct				:= HermesActIdle;
				bHermesWriteRetainLane1	:= FALSE;
			END_IF
		END_IF

	END_IF

	IF EDGENEG(p_bLinkOpsInvertStepInvert) THEN
		FOR i := 0 TO 200 DO
			IF (a_tyHermesBrdAvlData[1].a_tyXMLTableDataBrdAvl[i].sTitle = 'AT') THEN
				fConvertToLower_254(ADR(sLowerCase) , a_tyHermesBrdAvlData[1].a_tyXMLTableDataBrdAvl[i].sValue);

				IF (sLowerCase = 'flippedboard') THEN
					IF a_tyHermesBrdAvlData[1].a_tyXMLTableDataBrdAvl[i+1].sTitle = 'AV' THEN
						IF p_tyUSHermestyBoardAvailable.tyData.eFlippedBoard = 1 THEN
							a_tyHermesBrdAvlData[1].a_tyXMLTableDataBrdAvl[i+1].sValue	:= '2';
						ELSIF  p_tyUSHermestyBoardAvailable.tyData.eFlippedBoard = 2 THEN
							a_tyHermesBrdAvlData[1].a_tyXMLTableDataBrdAvl[i+1].sValue	:= '1';
						ELSE
							a_tyHermesBrdAvlData[1].a_tyXMLTableDataBrdAvl[i+1].sValue	:= '0';
						END_IF

						EXIT;

					END_IF

				END_IF

			END_IF
		END_FOR
	END_IF

END_ACTION
```

#### Cyclic.st - Do Not Change!!!
```iecst
(** 2019-05-04 **)
PROGRAM _CYCLIC

	IF bInitDone = FALSE THEN
		bInitDone	:= TRUE;

		Act_InitLocal;
		Act_InitGlobal;

	ELSIF bInitialDone = FALSE THEN
		IF p_bNtSettingsLoadDone = TRUE THEN
			bInitialDone	:= TRUE;

			Act_Initial;
		END_IF

	ELSE

		Act_RstErr;
		Act_LinkAction;
		Act_Action;
		Act_LinkEn;

		IF (p_bPrep = TRUE) AND (p_bEn = TRUE) AND (p_bDis = FALSE) THEN
			Act_Background_Route;
			Act_Link;
			Act_Background;
			Act_Main;
			Act_Background_Command;

		ELSE
			IF eStat <> HermesActIdle THEN
				eStatus	:= Done;
			ELSE
				eStatus	:= Idle;
			END_IF
		END_IF

		Act_Alarm;

	END_IF

END_PROGRAM
```

#### Act_RstErr.st - Do Not Change!!!
```iecst
(** 2019-05-04 **)
ACTION Act_RstErr:

	IF p_udiRstErr <> udiRstErrOld THEN
		bRstErr			:= TRUE;
		udiRstErrOld	:= p_udiRstErr;
	ELSE
		bRstErr			:= FALSE;
	END_IF

END_ACTION
```

#### Act_InitLocal.st - Do Not Change!!!
```iecst
(** 2019-05-04 **)
ACTION Act_InitLocal:

	//Input Reference Link To Local Variable
	p_eAct ACCESS ADR(eAct);
	p_udiRstErr ACCESS ADR(udiRstErr);
	p_bPrep ACCESS ADR(bPrep);
	p_bEn ACCESS ADR(bEn);
	p_bDis ACCESS ADR(bDis);
	pa_tyUSParam ACCESS ADR(a_tyUSParam);
	pa_tyDSParam ACCESS ADR(a_tyDSParam);
	p_tyRmtParam ACCESS ADR(tyRmtParam);
	p_tySvyParam ACCESS ADR(tySvyParam);
	p_tyRmtSetConfiguration ACCESS ADR(tyRmtSetConfiguration);
	p_tySvySetConfiguration ACCESS ADR(tySvySetConfiguration);

	p_bRmtPrep ACCESS ADR(bRmtPrep);
	p_bRmtEn ACCESS ADR(bRmtEn);
	p_bSvyPrep ACCESS ADR(bSvyPrep);
	p_bSvyEn ACCESS ADR(bSvyEn);
	p_sRetainFileName1 ACCESS ADR(sRetainFileName1);
	p_sRetainFileName2 ACCESS ADR(sRetainFileName2);
	p_sRetainFileName3 ACCESS ADR(sRetainFileName3);
	p_sRetainFileName4 ACCESS ADR(sRetainFileName4);
	p_udiRetainDataAddr1 ACCESS ADR(udiRetainDataAddr1);
	p_udiRetainDataLen1 ACCESS ADR(udiRetainDataLen1);
	p_udiRetainDataAddr2 ACCESS ADR(udiRetainDataAddr2);
	p_udiRetainDataLen2 ACCESS ADR(udiRetainDataLen2);
	p_udiRetainDataAddr3 ACCESS ADR(udiRetainDataAddr3);
	p_udiRetainDataLen3 ACCESS ADR(udiRetainDataLen3);
	p_udiRetainDataAddr4 ACCESS ADR(udiRetainDataAddr4);
	p_udiRetainDataLen4 ACCESS ADR(udiRetainDataLen4);

	p_sConfigFileName ACCESS ADR(sConfigFileName);
	p_sProgNm ACCESS ADR(sProgNm);
	p_bNtSettingsLoadDone ACCESS ADR(bNtSettingsLoadDone);
	p_bRmtHermesWriteConfig ACCESS ADR(bRmtHermesWriteConfig);
	p_bSvyHermesWriteConfig ACCESS ADR(bSvyHermesWriteConfig);
	p_bUISaveHMIConfigure ACCESS ADR(bUISaveHMIConfigure);
	p_bUISaveHMISvyConfig ACCESS ADR(bUISaveHMISvyConfig);
	p_sMcId ACCESS ADR(sMcId);

	p_bRmtFoundIndexUS1 ACCESS ADR(bRmtFoundIndexUS1);
	p_bRmtFoundIndexUS2 ACCESS ADR(bRmtFoundIndexUS2);
	p_bRmtFoundIndexUS3 ACCESS ADR(bRmtFoundIndexUS3);
	p_bRmtFoundIndexUS4 ACCESS ADR(bRmtFoundIndexUS4);
	p_bRmtFoundIndexDS1 ACCESS ADR(bRmtFoundIndexDS1);
	p_bRmtFoundIndexDS2 ACCESS ADR(bRmtFoundIndexDS2);
	p_bRmtFoundIndexDS3 ACCESS ADR(bRmtFoundIndexDS3);
	p_bRmtFoundIndexDS4 ACCESS ADR(bRmtFoundIndexDS4);
	p_udiRmtIndexUS1 ACCESS ADR(udiRmtIndexUS1);
	p_udiRmtIndexUS2 ACCESS ADR(udiRmtIndexUS2);
	p_udiRmtIndexUS3 ACCESS ADR(udiRmtIndexUS3);
	p_udiRmtIndexUS4 ACCESS ADR(udiRmtIndexUS4);
	p_udiRmtIndexDS1 ACCESS ADR(udiRmtIndexDS1);
	p_udiRmtIndexDS2 ACCESS ADR(udiRmtIndexDS2);
	p_udiRmtIndexDS3 ACCESS ADR(udiRmtIndexDS3);
	p_udiRmtIndexDS4 ACCESS ADR(udiRmtIndexDS4);

	p_bSvyFoundIndexUS1 ACCESS ADR(bSvyFoundIndexUS1);
	p_bSvyFoundIndexUS2 ACCESS ADR(bSvyFoundIndexUS2);
	p_bSvyFoundIndexUS3 ACCESS ADR(bSvyFoundIndexUS3);
	p_bSvyFoundIndexUS4 ACCESS ADR(bSvyFoundIndexUS4);
	p_bSvyFoundIndexDS1 ACCESS ADR(bSvyFoundIndexDS1);
	p_bSvyFoundIndexDS2 ACCESS ADR(bSvyFoundIndexDS2);
	p_bSvyFoundIndexDS3 ACCESS ADR(bSvyFoundIndexDS3);
	p_bSvyFoundIndexDS4 ACCESS ADR(bSvyFoundIndexDS4);

	p_udiSvyIndexUS1 ACCESS ADR(udiSvyIndexUS1);
	p_udiSvyIndexUS2 ACCESS ADR(udiSvyIndexUS2);
	p_udiSvyIndexUS3 ACCESS ADR(udiSvyIndexUS3);
	p_udiSvyIndexUS4 ACCESS ADR(udiSvyIndexUS4);
	p_udiSvyIndexDS1 ACCESS ADR(udiSvyIndexDS1);
	p_udiSvyIndexDS2 ACCESS ADR(udiSvyIndexDS2);
	p_udiSvyIndexDS3 ACCESS ADR(udiSvyIndexDS3);
	p_udiSvyIndexDS4 ACCESS ADR(udiSvyIndexDS4);

	p_bReverseReceiveRoute ACCESS ADR(bReverseReceiveRoute);
	p_bReverseSentRoute ACCESS ADR(bReverseSendRoute);

	p_bManualRmvRoute ACCESS ADR(bManualRmvRoute);
	p_bReturnRoute ACCESS ADR(bReturnRoute);
	p_bNomRouteEn ACCESS ADR(bNomRouteEn);
END_ACTION
```

#### Act_Initial.st - Do Not Change!!!
```iecst
(** 2019-05-04 **)
ACTION Act_Initial:
	//Initial

	//Retain Data
	p_udiRetainDataAddr1	:= ADR(a_tyHermesBrdAvlData);
	p_udiRetainDataLen1	:= SIZEOF(a_tyHermesBrdAvlData);

	sStatTxt	:= a_sStatText[eStat];

	fbDirCreate1.sDevice	:= 'F';
	fbDirCreate1.sDirName	:= 'User';
	fbDirCreate1(bEn := FALSE);

	fbDirCreate2.sDevice	:= 'User';
	fbDirCreate2.sDirName	:= 'Retain';
	fbDirCreate2(bEn := FALSE);

	fbDirCreate3.sDevice	:= 'User';
	fbDirCreate3.sDirName	:= 'Log';
	fbDirCreate3(bEn := FALSE);

	fbDirCreate4.sDevice	:= 'User';
	fbDirCreate4.sDirName	:= 'MachineParameter';
	fbDirCreate4(bEn := FALSE);

	fbFileRead1.sDevice			:= 'McParam';
	fbFileRead1.sFile			:= p_sConfigFileName;
	fbFileRead1.udiOffset		:= 0;
	fbFileRead1.p_Dest			:= ADR(tyCurrConfiguration);
	fbFileRead1.udiLen			:= SIZEOF(tyCurrConfiguration);
	fbFileRead1(bEn := FALSE);

	fbFileWrite1.sDevice		:= 'McParam';
	fbFileWrite1.sFile			:= p_sConfigFileName;
	fbFileWrite1.udiOffset		:= 0;
	fbFileWrite1.p_Src			:= ADR(tyConfigurationWr);
	fbFileWrite1.udiLen			:= SIZEOF(tyConfigurationWr);
	fbFileWrite1.udiOption		:= 0;
	fbFileWrite1(bEn := FALSE);

	fbFileRead2.sDevice			:= 'Retain';
	fbFileRead2.sFile			:= p_sRetainFileName1;
	fbFileRead2.udiOffset		:= 0;
	fbFileRead2.p_Dest			:= p_udiRetainDataAddr1;
	fbFileRead2.udiLen			:= p_udiRetainDataLen1;
	fbFileRead2(bEn := FALSE);

	fbFileWrite2.sDevice		:= 'Retain';
	fbFileWrite2.sFile			:= p_sRetainFileName1;
	fbFileWrite2.udiOffset		:= 0;
	fbFileWrite2.p_Src			:= p_udiRetainDataAddr1;
	fbFileWrite2.udiLen			:= p_udiRetainDataLen1;
	fbFileWrite2.udiOption		:= 0;
	fbFileWrite2(bEn := FALSE);

	fbFileRead3.sDevice			:= 'Retain';
	fbFileRead3.sFile			:= p_sRetainFileName2;
	fbFileRead3.udiOffset		:= 0;
	fbFileRead3.p_Dest			:= p_udiRetainDataAddr2;
	fbFileRead3.udiLen			:= p_udiRetainDataLen2;
	fbFileRead3(bEn := FALSE);

	fbFileWrite3.sDevice		:= 'Retain';
	fbFileWrite3.sFile			:= p_sRetainFileName2;
	fbFileWrite3.udiOffset		:= 0;
	fbFileWrite3.udiOption		:= 0;
	fbFileWrite3.p_Src			:= p_udiRetainDataAddr2;
	fbFileWrite3.udiLen			:= p_udiRetainDataLen2;
	fbFileWrite3(bEn := FALSE);

	fbFileRead4.sDevice			:= 'Retain';
	fbFileRead4.sFile			:= p_sRetainFileName3;
	fbFileRead4.udiOffset		:= 0;
	fbFileRead4.p_Dest			:= p_udiRetainDataAddr3;
	fbFileRead4.udiLen			:= p_udiRetainDataLen3;
	fbFileRead4(bEn := FALSE);

	fbFileWrite4.sDevice		:= 'Retain';
	fbFileWrite4.sFile			:= p_sRetainFileName3;
	fbFileWrite4.udiOffset		:= 0;
	fbFileWrite4.udiOption		:= 0;
	fbFileWrite4.p_Src			:= p_udiRetainDataAddr3;
	fbFileWrite4.udiLen			:= p_udiRetainDataLen3;
	fbFileWrite4(bEn := FALSE);

	fbFileRead5.sDevice			:= 'Retain';
	fbFileRead5.sFile			:= p_sRetainFileName4;
	fbFileRead5.udiOffset		:= 0;
	fbFileRead5.p_Dest			:= p_udiRetainDataAddr4;
	fbFileRead5.udiLen			:= p_udiRetainDataLen4;
	fbFileRead5(bEn := FALSE);

	fbFileWrite5.sDevice		:= 'Retain';
	fbFileWrite5.sFile			:= p_sRetainFileName4;
	fbFileWrite5.udiOffset		:= 0;
	fbFileWrite5.udiOption		:= 0;
	fbFileWrite5.p_Src			:= p_udiRetainDataAddr4;
	fbFileWrite5.udiLen			:= p_udiRetainDataLen4;
	fbFileWrite5(bEn := FALSE);

	//Command
	memset(ADR(a_tyCommandProcessList),0,SIZEOF(a_tyCommandProcessList));
	usiProcessCmdBffr := 0;
	usiUSIdent  := fHermesAddOneCommandGate(TRUE,p_USHermesCommandParam,ADR(tyCurrConfiguration.a_tyUSParam[0].sUpstreamInterfaceId),p_McParamUSCommMod,ADR(a_tyCommandProcessList),ADR(usiProcessCmdBffr));
	usiDSIdent  := fHermesAddOneCommandGate(FALSE,p_DSHermesCommandParam,ADR(tyCurrConfiguration.a_tyDSParam[0].sDownstreamInterfaceId),p_McParamDSCommMod,ADR(a_tyCommandProcessList),ADR(usiProcessCmdBffr));
	usiUSIdent2 := fHermesAddOneCommandGate(TRUE,p_USHermes2CommandParam,ADR(tyCurrConfiguration.a_tyUSParam[1].sUpstreamInterfaceId),p_McParamUSComm2Mod,ADR(a_tyCommandProcessList),ADR(usiProcessCmdBffr));

	//output
	bCmdInitialCompl := TRUE;

	//tyCurrConfiguration
	//Feature(Machine Safety)
	p_HermesUSCmdFeaturePause := ADR(tyCurrConfiguration.a_tyUSParam[0].bFeatureCommand);
	p_HermesUSCmdPause := ADR(a_tyCommandPause[usiUSIdent]);
	p_HermesDSCmdFeaturePause := ADR(tyCurrConfiguration.a_tyDSParam[0].bFeatureCommand);
	p_HermesDSCmdPause := ADR(a_tyCommandPause[usiDSIdent]);
	a_tyCommandPause[usiUSIdent].bFeatureRequestFrom :=  p_bNTParamMachineSafetySig;
	a_tyCommandPause[usiUSIdent].bFeatureRequestTo   :=  p_bNTParamUnlockCovPrep;

	a_tyCommandPause[usiDSIdent].bFeatureRequestFrom := p_bNTParamMachineSafetySig;
	a_tyCommandPause[usiDSIdent].bFeatureRequestTo	:=  p_bNTParamUnlockCovPrep;

	//Feature(Oven Info)
	//p_HermesUSCmdFeaturePause := ADR(tyCurrConfiguration.a_tyUSParam[1].bFeatureCommand);
	//p_HermesUSCmdPause := ADR(a_tyCommandPause[usiUSIdent2]);
	//a_tyCommandLockInputConv[usiUSIdent].bFeatureLockConvTo   :=  p_bNTParamOvenInfoAPrep;
	//a_tyCommandLockInputConv[usiDSIdent].bFeatureLockConvFrom := p_bNTParamOvenInfoAPrep;
	//a_tyCommandLockInputConv[usiUSIdent2].bFeatureLockConvTo  :=  p_bNTParamOvenInfoBPrep;

END_ACTION
```

#### Act_Main.st - Do Not Change!!!
```iecst
(** 2021-08-01 **)
ACTION Act_Main:

	IF eStatOld <> eStat THEN
		fbDirCreate1(bEn := FALSE);
		fbDirCreate2(bEn := FALSE);
		fbDirCreate3(bEn := FALSE);
		fbDirCreate4(bEn := FALSE);
		fbFileRead1(bEn := FALSE);
		fbFileWrite1(bEn := FALSE);
		fbFileRead2(bEn := FALSE);
		fbFileWrite2(bEn := FALSE);
		fbFileRead3(bEn := FALSE);
		fbFileWrite3(bEn := FALSE);
		fbFileRead4(bEn := FALSE);
		fbFileWrite4(bEn := FALSE);
		fbFileRead5(bEn := FALSE);
		fbFileWrite5(bEn := FALSE);
		usiStep			:= 0;
		bFileNotFound	:= FALSE;

		sStatTxt	:= a_sStatText[eStat];

		eStatOld	:= eStat;

		eStatus		:= Busy;
	END_IF

	//Main
	CASE eStat OF

		HermesActIdle:
			eStatus	:= Idle;

		HermesActCreateDir:
			IF eStatus = Idle OR eStatus = Busy THEN

				eStatus	:= Busy;

				CASE usiStep OF
					0:
						fbDirCreate1(bEn := TRUE);
						IF fbDirCreate1.udiStatus = 0 THEN
							usiStep	:= 1;
						ELSIF fbDirCreate1.udiStatus < 65534 THEN
							eStatus		:= Error;

							IF fbDirCreate1.udiStatus = 1908 THEN
								udiStatus	:= 10000;	//Create User Directory Error
							ELSE
								udiStatus	:= fbDirCreate1.udiStatus;
							END_IF
						END_IF

					1:
						fbDirCreate2(bEn := TRUE);
						IF fbDirCreate2.udiStatus = 0 THEN
							usiStep	:= 2;
						ELSIF fbDirCreate2.udiStatus < 65534 THEN
							eStatus		:= Error;

							IF fbDirCreate2.udiStatus = 1908 THEN
								udiStatus	:= 10001;	//Create Retain Directory Error
							ELSE
								udiStatus	:= fbDirCreate2.udiStatus;
							END_IF
						END_IF

					2:
						fbDirCreate3(bEn := TRUE);
						IF fbDirCreate3.udiStatus = 0 THEN
							usiStep	:= 3;
						ELSIF fbDirCreate3.udiStatus < 65534 THEN
							eStatus		:= Error;

							IF fbDirCreate3.udiStatus = 1908 THEN
								udiStatus	:= 10010;	//Create Log Directory Error
							ELSE
								udiStatus	:= fbDirCreate3.udiStatus;
							END_IF
						END_IF

					3:
						fbDirCreate4(bEn := TRUE);
						IF fbDirCreate4.udiStatus = 0 THEN
							eStatus	:= Done;
						ELSIF fbDirCreate4.udiStatus < 65534 THEN
							eStatus		:= Error;

							IF fbDirCreate4.udiStatus = 1908 THEN
								udiStatus	:= 10011;	//Create Machine Parameter Directory Error
							ELSE
								udiStatus	:= fbDirCreate4.udiStatus;
							END_IF
						END_IF

				END_CASE

			END_IF

		HermesActReadRetainLane1:
			IF eStatus = Idle OR eStatus = Busy THEN

				eStatus	:= Busy;

				fbFileRead2(bEn := TRUE);

				IF fbFileRead2.udiStatus = 0 THEN
					eStatus	:= Done;
				ELSIF fbFileRead2.udiStatus < 65534 THEN
					eStatus	:= Error;

					IF fbFileRead2.udiStatus = 1900 THEN
						udiStatus	:= 10002;	//File Open Error While Reading Retain File
					ELSIF fbFileRead2.udiStatus = 1902 THEN
						udiStatus	:= 10003;	//File Read Error While Reading Retain File
					ELSIF fbFileRead2.udiStatus = 1904 THEN
						udiStatus	:= 10004;	//File Close Error While Reading Retain File
					ELSIF fbFileRead2.udiStatus = 1915 THEN
						eStatus			:= Done;
						bFileNotFound	:= TRUE;
					ELSE
						udiStatus	:= fbFileRead2.udiStatus;
					END_IF
				END_IF

			END_IF

		HermesActWriteRetainLane1:
			IF eStatus = Idle OR eStatus = Busy THEN

				eStatus	:= Busy;

				fbFileWrite2(bEn := TRUE);

				IF fbFileWrite2.udiStatus = 0 THEN
					eStatus	:= Done;
				ELSIF fbFileWrite2.udiStatus < 65534 THEN
					eStatus	:= Error;

					IF fbFileWrite2.udiStatus = 1900 THEN
						udiStatus	:= 10005;	//File Open Error While Writing Retain File
					ELSIF fbFileWrite2.udiStatus = 1901 THEN
						udiStatus	:= 10006;	//File Create Error While Writing Retain File
					ELSIF fbFileWrite2.udiStatus = 1903 THEN
						udiStatus	:= 10007;	//File Write Error While Writing Retain File
					ELSIF fbFileWrite2.udiStatus = 1904 THEN
						udiStatus	:= 10008;	//File Close Error While Writing Retain File
					ELSIF fbFileWrite2.udiStatus = 1914 THEN
						udiStatus	:= 10009;	//Directory Does Not Exist While Writing Retain File
					ELSE
						udiStatus	:= fbFileWrite2.udiStatus;
					END_IF
				END_IF

			END_IF

		HermesActReadRetainLane2:
			IF eStatus = Idle OR eStatus = Busy THEN

				eStatus	:= Busy;

				fbFileRead3(bEn := TRUE);

				IF fbFileRead3.udiStatus = 0 THEN
					eStatus	:= Done;
				ELSIF fbFileRead3.udiStatus < 65534 THEN
					eStatus	:= Error;

					IF fbFileRead3.udiStatus = 1900 THEN
						udiStatus	:= 10032;	//File Open Error While Reading Retain File
					ELSIF fbFileRead3.udiStatus = 1902 THEN
						udiStatus	:= 10033;	//File Read Error While Reading Retain File
					ELSIF fbFileRead3.udiStatus = 1904 THEN
						udiStatus	:= 10034;	//File Close Error While Reading Retain File
					ELSIF fbFileRead3.udiStatus = 1915 THEN
						eStatus			:= Done;
						bFileNotFound	:= TRUE;
					ELSE
						udiStatus	:= fbFileRead3.udiStatus;
					END_IF
				END_IF

			END_IF

		HermesActWriteRetainLane2:
			IF eStatus = Idle OR eStatus = Busy THEN

				eStatus	:= Busy;

				fbFileWrite3(bEn := TRUE);

				IF fbFileWrite3.udiStatus = 0 THEN
					eStatus	:= Done;
				ELSIF fbFileWrite3.udiStatus < 65534 THEN
					eStatus	:= Error;

					IF fbFileWrite3.udiStatus = 1900 THEN
						udiStatus	:= 10035;	//File Open Error While Writing Retain File
					ELSIF fbFileWrite3.udiStatus = 1901 THEN
						udiStatus	:= 10036;	//File Create Error While Writing Retain File
					ELSIF fbFileWrite3.udiStatus = 1903 THEN
						udiStatus	:= 10037;	//File Write Error While Writing Retain File
					ELSIF fbFileWrite3.udiStatus = 1904 THEN
						udiStatus	:= 10038;	//File Close Error While Writing Retain File
					ELSIF fbFileWrite3.udiStatus = 1914 THEN
						udiStatus	:= 10039;	//Directory Does Not Exist While Writing Retain File
					ELSE
						udiStatus	:= fbFileWrite3.udiStatus;
					END_IF
				END_IF

			END_IF

		HermesActReadRetainLane3:
			IF eStatus = Idle OR eStatus = Busy THEN

				eStatus	:= Busy;

				fbFileRead4(bEn := TRUE);

				IF fbFileRead4.udiStatus = 0 THEN
					eStatus	:= Done;
				ELSIF fbFileRead4.udiStatus < 65534 THEN
					eStatus	:= Error;

					IF fbFileRead4.udiStatus = 1900 THEN
						udiStatus	:= 10042;	//File Open Error While Reading Retain File
					ELSIF fbFileRead4.udiStatus = 1902 THEN
						udiStatus	:= 10043;	//File Read Error While Reading Retain File
					ELSIF fbFileRead4.udiStatus = 1904 THEN
						udiStatus	:= 10044;	//File Close Error While Reading Retain File
					ELSIF fbFileRead4.udiStatus = 1915 THEN
						eStatus			:= Done;
						bFileNotFound	:= TRUE;
					ELSE
						udiStatus	:= fbFileRead4.udiStatus;
					END_IF
				END_IF

			END_IF

		HermesActWriteRetainLane3:
			IF eStatus = Idle OR eStatus = Busy THEN

				eStatus	:= Busy;

				fbFileWrite4(bEn := TRUE);

				IF fbFileWrite4.udiStatus = 0 THEN
					eStatus	:= Done;
				ELSIF fbFileWrite4.udiStatus < 65534 THEN
					eStatus	:= Error;

					IF fbFileWrite4.udiStatus = 1900 THEN
						udiStatus	:= 10045;	//File Open Error While Writing Retain File
					ELSIF fbFileWrite4.udiStatus = 1901 THEN
						udiStatus	:= 10046;	//File Create Error While Writing Retain File
					ELSIF fbFileWrite4.udiStatus = 1903 THEN
						udiStatus	:= 10047;	//File Write Error While Writing Retain File
					ELSIF fbFileWrite4.udiStatus = 1904 THEN
						udiStatus	:= 10048;	//File Close Error While Writing Retain File
					ELSIF fbFileWrite4.udiStatus = 1914 THEN
						udiStatus	:= 10049;	//Directory Does Not Exist While Writing Retain File
					ELSE
						udiStatus	:= fbFileWrite4.udiStatus;
					END_IF
				END_IF

			END_IF

		HermesActReadRetainLane4:
			IF eStatus = Idle OR eStatus = Busy THEN

				eStatus	:= Busy;

				fbFileRead5(bEn := TRUE);

				IF fbFileRead5.udiStatus = 0 THEN
					eStatus	:= Done;
				ELSIF fbFileRead5.udiStatus < 65534 THEN
					eStatus	:= Error;

					IF fbFileRead5.udiStatus = 1900 THEN
						udiStatus	:= 10052;	//File Open Error While Reading Retain File
					ELSIF fbFileRead5.udiStatus = 1902 THEN
						udiStatus	:= 10053;	//File Read Error While Reading Retain File
					ELSIF fbFileRead5.udiStatus = 1904 THEN
						udiStatus	:= 10054;	//File Close Error While Reading Retain File
					ELSIF fbFileRead5.udiStatus = 1915 THEN
						eStatus			:= Done;
						bFileNotFound	:= TRUE;
					ELSE
						udiStatus	:= fbFileRead5.udiStatus;
					END_IF
				END_IF

			END_IF

		HermesActWriteRetainLane4:
			IF eStatus = Idle OR eStatus = Busy THEN

				eStatus	:= Busy;

				fbFileWrite5(bEn := TRUE);

				IF fbFileWrite5.udiStatus = 0 THEN
					eStatus	:= Done;
				ELSIF fbFileWrite5.udiStatus < 65534 THEN
					eStatus	:= Error;

					IF fbFileWrite5.udiStatus = 1900 THEN
						udiStatus	:= 10055;	//File Open Error While Writing Retain File
					ELSIF fbFileWrite5.udiStatus = 1901 THEN
						udiStatus	:= 10056;	//File Create Error While Writing Retain File
					ELSIF fbFileWrite5.udiStatus = 1903 THEN
						udiStatus	:= 10057;	//File Write Error While Writing Retain File
					ELSIF fbFileWrite5.udiStatus = 1904 THEN
						udiStatus	:= 10058;	//File Close Error While Writing Retain File
					ELSIF fbFileWrite5.udiStatus = 1914 THEN
						udiStatus	:= 10059;	//Directory Does Not Exist While Writing Retain File
					ELSE
						udiStatus	:= fbFileWrite5.udiStatus;
					END_IF
				END_IF

			END_IF

		HermesActReadConfig:
			IF eStatus = Idle OR eStatus = Busy THEN

				eStatus	:= Busy;

				fbFileRead1(bEn := TRUE);

				IF fbFileRead1.udiStatus = 0 THEN
					eStatus	:= Done;
					tyConfigurationWr := tyCurrConfiguration;
				ELSIF fbFileRead1.udiStatus < 65534 THEN
					eStatus	:= Error;

					IF fbFileRead1.udiStatus = 1900 THEN
						udiStatus	:= 10012;	//File Open Error While Reading Config File
					ELSIF fbFileRead1.udiStatus = 1902 THEN
						udiStatus	:= 10013;	//File Read Error While Reading Config File
					ELSIF fbFileRead1.udiStatus = 1904 THEN
						udiStatus	:= 10014;	//File Close Error While Reading Config File
					ELSIF fbFileRead1.udiStatus = 1915 THEN
						eStatus			:= Done;
						bFileNotFound	:= TRUE;
					ELSE
						udiStatus	:= fbFileRead1.udiStatus;
					END_IF
				END_IF

			END_IF

		HermesActWriteConfig:
			IF eStatus = Idle OR eStatus = Busy THEN

				eStatus	:= Busy;

				fbFileWrite1(bEn := TRUE);

				IF fbFileWrite1.udiStatus = 0 THEN
					eStatus	:= Done;
					tyCurrConfiguration := tyConfigurationWr;
				ELSIF fbFileWrite1.udiStatus < 65534 THEN
					eStatus	:= Error;

					IF fbFileWrite1.udiStatus = 1900 THEN
						udiStatus	:= 10015;	//File Open Error While Writing Config File
					ELSIF fbFileWrite1.udiStatus = 1901 THEN
						udiStatus	:= 10016;	//File Create Error While Writing Config File
					ELSIF fbFileWrite1.udiStatus = 1903 THEN
						udiStatus	:= 10017;	//File Write Error While Writing Config File
					ELSIF fbFileWrite1.udiStatus = 1904 THEN
						udiStatus	:= 10018;	//File Close Error While Writing Config File
					ELSIF fbFileWrite1.udiStatus = 1914 THEN
						udiStatus	:= 10019;	//Directory Does Not Exist While Writing Config File
					ELSE
						udiStatus	:= fbFileWrite1.udiStatus;
					END_IF
				END_IF

			END_IF

		ELSE
			IF eStatus = Idle OR eStatus = Busy THEN
				eStatus	:= Done;
			END_IF

	END_CASE

END_ACTION
```

#### Act_Background.st - Do Not Change!!!
```iecst
(** 2021-08-01 **)
ACTION Act_Background:

	//Update Configuration

	IF p_bSvyPrep = TRUE AND p_bSvyEn = TRUE AND p_bSvyHermesWriteConfig THEN

		IF p_bSvyFoundIndexUS1 THEN
			tyConfigurationWr.a_tyUSParam[0].iLaneID		            := p_tySvySetConfiguration.tyData.a_tyUpstreamConfigurations[0].iUpstreamLaneId;		//change from p_udiSvyIndexUS1
			tyConfigurationWr.a_tyUSParam[0].sHostAddress           	:= p_tySvySetConfiguration.tyData.a_tyUpstreamConfigurations[0].sHostAddress;			//
			tyConfigurationWr.a_tyUSParam[0].uiHostPort	                := p_tySvySetConfiguration.tyData.a_tyUpstreamConfigurations[0].uiPort;					//
			tyConfigurationWr.a_tyUSParam[0].sUpstreamInterfaceId   	:= p_tySvySetConfiguration.tyData.a_tyUpstreamConfigurations[0].sUpstreamInterfaceId;	//
		END_IF

		IF p_bSvyFoundIndexUS2 THEN
			tyConfigurationWr.a_tyUSParam[1].iLaneID		            := p_tySvySetConfiguration.tyData.a_tyUpstreamConfigurations[1].iUpstreamLaneId;		//change from p_udiSvyIndexUS2
			tyConfigurationWr.a_tyUSParam[1].sHostAddress           	:= p_tySvySetConfiguration.tyData.a_tyUpstreamConfigurations[1].sHostAddress;			//
			tyConfigurationWr.a_tyUSParam[1].uiHostPort	                := p_tySvySetConfiguration.tyData.a_tyUpstreamConfigurations[1].uiPort;					//
			tyConfigurationWr.a_tyUSParam[1].sUpstreamInterfaceId   	:= p_tySvySetConfiguration.tyData.a_tyUpstreamConfigurations[1].sUpstreamInterfaceId;	//
		END_IF

		IF p_bSvyFoundIndexUS3 THEN
			tyConfigurationWr.a_tyUSParam[2].iLaneID		            := p_tySvySetConfiguration.tyData.a_tyUpstreamConfigurations[2].iUpstreamLaneId;		//change from p_udiSvyIndexUS3
			tyConfigurationWr.a_tyUSParam[2].sHostAddress           	:= p_tySvySetConfiguration.tyData.a_tyUpstreamConfigurations[2].sHostAddress;			//
			tyConfigurationWr.a_tyUSParam[2].uiHostPort	                := p_tySvySetConfiguration.tyData.a_tyUpstreamConfigurations[2].uiPort;					//
			tyConfigurationWr.a_tyUSParam[2].sUpstreamInterfaceId   	:= p_tySvySetConfiguration.tyData.a_tyUpstreamConfigurations[2].sUpstreamInterfaceId;	//
		END_IF

		IF p_bSvyFoundIndexUS4 THEN
			tyConfigurationWr.a_tyUSParam[3].iLaneID		            := p_tySvySetConfiguration.tyData.a_tyUpstreamConfigurations[3].iUpstreamLaneId;		//change from p_udiSvyIndexUS4
			tyConfigurationWr.a_tyUSParam[3].sHostAddress           	:= p_tySvySetConfiguration.tyData.a_tyUpstreamConfigurations[3].sHostAddress;			//
			tyConfigurationWr.a_tyUSParam[3].uiHostPort	                := p_tySvySetConfiguration.tyData.a_tyUpstreamConfigurations[3].uiPort;					//
			tyConfigurationWr.a_tyUSParam[3].sUpstreamInterfaceId   	:= p_tySvySetConfiguration.tyData.a_tyUpstreamConfigurations[3].sUpstreamInterfaceId;	//
		END_IF

		IF p_bSvyFoundIndexDS1 THEN
			tyConfigurationWr.a_tyDSParam[0].iLaneID	            	:= p_tySvySetConfiguration.tyData.a_tyDownstreamConfigurations[0].iDownstreamLaneId;		//change from p_udiSvyIndexDS1
			tyConfigurationWr.a_tyDSParam[0].uiSvrPort               	:= p_tySvySetConfiguration.tyData.a_tyDownstreamConfigurations[0].uiPort;					//
			tyConfigurationWr.a_tyDSParam[0].sDownstreamInterfaceId  	:= p_tySvySetConfiguration.tyData.a_tyDownstreamConfigurations[0].sDownstreamInterfaceId;	//
		END_IF

		IF p_bSvyFoundIndexDS2 THEN
			tyConfigurationWr.a_tyDSParam[1].iLaneID	            	:= p_tySvySetConfiguration.tyData.a_tyDownstreamConfigurations[1].iDownstreamLaneId;		//change from p_udiSvyIndexDS2
			tyConfigurationWr.a_tyDSParam[1].uiSvrPort               	:= p_tySvySetConfiguration.tyData.a_tyDownstreamConfigurations[1].uiPort;					//
			tyConfigurationWr.a_tyDSParam[1].sDownstreamInterfaceId  	:= p_tySvySetConfiguration.tyData.a_tyDownstreamConfigurations[1].sDownstreamInterfaceId;	//
		END_IF

		IF p_bSvyFoundIndexDS3 THEN
			tyConfigurationWr.a_tyDSParam[2].iLaneID	            	:= p_tySvySetConfiguration.tyData.a_tyDownstreamConfigurations[2].iDownstreamLaneId;		//change from p_udiSvyIndexDS3
			tyConfigurationWr.a_tyDSParam[2].uiSvrPort               	:= p_tySvySetConfiguration.tyData.a_tyDownstreamConfigurations[2].uiPort;					//
			tyConfigurationWr.a_tyDSParam[2].sDownstreamInterfaceId  	:= p_tySvySetConfiguration.tyData.a_tyDownstreamConfigurations[2].sDownstreamInterfaceId;	//
		END_IF

		IF p_bSvyFoundIndexDS4 THEN
			tyConfigurationWr.a_tyDSParam[3].iLaneID	            	:= p_tySvySetConfiguration.tyData.a_tyDownstreamConfigurations[3].iDownstreamLaneId;		//change from p_udiSvyIndexDS4
			tyConfigurationWr.a_tyDSParam[3].uiSvrPort               	:= p_tySvySetConfiguration.tyData.a_tyDownstreamConfigurations[3].uiPort;					//
			tyConfigurationWr.a_tyDSParam[3].sDownstreamInterfaceId  	:= p_tySvySetConfiguration.tyData.a_tyDownstreamConfigurations[3].sDownstreamInterfaceId;	//
		END_IF

		IF p_tySvySetConfiguration.tyAvl.bMachineId = TRUE THEN

			tyConfigurationWr.a_tyUSParam[0].sMachineId		:= p_tySvySetConfiguration.tyData.sMachineId;
			tyConfigurationWr.a_tyDSParam[0].sMachineId		:= p_tySvySetConfiguration.tyData.sMachineId;
			tyConfigurationWr.tySvyParam.sMachineId		    := p_tySvySetConfiguration.tyData.sMachineId;

		END_IF

		IF p_tySvySetConfiguration.tyAvl.bSupervisorySystemPort = TRUE THEN

			tyConfigurationWr.tySvyParam.uiSvySvstemPort	:= p_tySvySetConfiguration.tyData.uiSupervisorySystemPort;

		END_IF

	ELSIF p_bRmtPrep = TRUE AND p_bRmtEn = TRUE AND p_bRmtHermesWriteConfig THEN

		IF p_bRmtFoundIndexUS1 THEN
			tyConfigurationWr.a_tyUSParam[0].iLaneID		            := p_tyRmtSetConfiguration.tyData.a_tyUpstreamConfigurations[p_udiRmtIndexUS1].iUpstreamLaneId;
			tyConfigurationWr.a_tyUSParam[0].sHostAddress           	:= p_tyRmtSetConfiguration.tyData.a_tyUpstreamConfigurations[p_udiRmtIndexUS1].sHostAddress;
			tyConfigurationWr.a_tyUSParam[0].uiHostPort	                := p_tyRmtSetConfiguration.tyData.a_tyUpstreamConfigurations[p_udiRmtIndexUS1].uiPort;
			tyConfigurationWr.a_tyUSParam[0].sUpstreamInterfaceId   	:= p_tyRmtSetConfiguration.tyData.a_tyUpstreamConfigurations[p_udiRmtIndexUS1].sUpstreamInterfaceId;
		END_IF

		IF p_bRmtFoundIndexUS2 THEN
			tyConfigurationWr.a_tyUSParam[1].iLaneID		            := p_tyRmtSetConfiguration.tyData.a_tyUpstreamConfigurations[p_udiRmtIndexUS2].iUpstreamLaneId;
			tyConfigurationWr.a_tyUSParam[1].sHostAddress           	:= p_tyRmtSetConfiguration.tyData.a_tyUpstreamConfigurations[p_udiRmtIndexUS2].sHostAddress;
			tyConfigurationWr.a_tyUSParam[1].uiHostPort	                := p_tyRmtSetConfiguration.tyData.a_tyUpstreamConfigurations[p_udiRmtIndexUS2].uiPort;
			tyConfigurationWr.a_tyUSParam[1].sUpstreamInterfaceId   	:= p_tyRmtSetConfiguration.tyData.a_tyUpstreamConfigurations[p_udiRmtIndexUS2].sUpstreamInterfaceId;
		END_IF

		IF p_bRmtFoundIndexUS3 THEN
			tyConfigurationWr.a_tyUSParam[2].iLaneID		            := p_tyRmtSetConfiguration.tyData.a_tyUpstreamConfigurations[p_udiRmtIndexUS3].iUpstreamLaneId;
			tyConfigurationWr.a_tyUSParam[2].sHostAddress           	:= p_tyRmtSetConfiguration.tyData.a_tyUpstreamConfigurations[p_udiRmtIndexUS3].sHostAddress;
			tyConfigurationWr.a_tyUSParam[2].uiHostPort	                := p_tyRmtSetConfiguration.tyData.a_tyUpstreamConfigurations[p_udiRmtIndexUS3].uiPort;
			tyConfigurationWr.a_tyUSParam[2].sUpstreamInterfaceId   	:= p_tyRmtSetConfiguration.tyData.a_tyUpstreamConfigurations[p_udiRmtIndexUS3].sUpstreamInterfaceId;
		END_IF

		IF p_bRmtFoundIndexUS4 THEN
			tyConfigurationWr.a_tyUSParam[3].iLaneID		            := p_tyRmtSetConfiguration.tyData.a_tyUpstreamConfigurations[p_udiRmtIndexUS4].iUpstreamLaneId;
			tyConfigurationWr.a_tyUSParam[3].sHostAddress           	:= p_tyRmtSetConfiguration.tyData.a_tyUpstreamConfigurations[p_udiRmtIndexUS4].sHostAddress;
			tyConfigurationWr.a_tyUSParam[3].uiHostPort	                := p_tyRmtSetConfiguration.tyData.a_tyUpstreamConfigurations[p_udiRmtIndexUS4].uiPort;
			tyConfigurationWr.a_tyUSParam[3].sUpstreamInterfaceId   	:= p_tyRmtSetConfiguration.tyData.a_tyUpstreamConfigurations[p_udiRmtIndexUS4].sUpstreamInterfaceId;
		END_IF

		IF p_bRmtFoundIndexDS1 THEN
			tyConfigurationWr.a_tyDSParam[0].iLaneID	            	:= p_tyRmtSetConfiguration.tyData.a_tyDownstreamConfigurations[p_udiRmtIndexDS1].iDownstreamLaneId;
			tyConfigurationWr.a_tyDSParam[0].uiSvrPort               	:= p_tyRmtSetConfiguration.tyData.a_tyDownstreamConfigurations[p_udiRmtIndexDS1].uiPort;
			tyConfigurationWr.a_tyDSParam[0].sDownstreamInterfaceId  	:= p_tyRmtSetConfiguration.tyData.a_tyDownstreamConfigurations[p_udiRmtIndexDS1].sDownstreamInterfaceId;
		END_IF

		IF p_bRmtFoundIndexDS2 THEN
			tyConfigurationWr.a_tyDSParam[1].iLaneID	            	:= p_tyRmtSetConfiguration.tyData.a_tyDownstreamConfigurations[p_udiRmtIndexDS2].iDownstreamLaneId;
			tyConfigurationWr.a_tyDSParam[1].uiSvrPort               	:= p_tyRmtSetConfiguration.tyData.a_tyDownstreamConfigurations[p_udiRmtIndexDS2].uiPort;
			tyConfigurationWr.a_tyDSParam[1].sDownstreamInterfaceId  	:= p_tyRmtSetConfiguration.tyData.a_tyDownstreamConfigurations[p_udiRmtIndexDS2].sDownstreamInterfaceId;
		END_IF

		IF p_bRmtFoundIndexDS3 THEN
			tyConfigurationWr.a_tyDSParam[2].iLaneID	            	:= p_tyRmtSetConfiguration.tyData.a_tyDownstreamConfigurations[p_udiRmtIndexDS3].iDownstreamLaneId;
			tyConfigurationWr.a_tyDSParam[2].uiSvrPort               	:= p_tyRmtSetConfiguration.tyData.a_tyDownstreamConfigurations[p_udiRmtIndexDS3].uiPort;
			tyConfigurationWr.a_tyDSParam[2].sDownstreamInterfaceId  	:= p_tyRmtSetConfiguration.tyData.a_tyDownstreamConfigurations[p_udiRmtIndexDS3].sDownstreamInterfaceId;
		END_IF

		IF p_bRmtFoundIndexDS4 THEN
			tyConfigurationWr.a_tyDSParam[3].iLaneID	            	:= p_tyRmtSetConfiguration.tyData.a_tyDownstreamConfigurations[p_udiRmtIndexDS4].iDownstreamLaneId;
			tyConfigurationWr.a_tyDSParam[3].uiSvrPort               	:= p_tyRmtSetConfiguration.tyData.a_tyDownstreamConfigurations[p_udiRmtIndexDS4].uiPort;
			tyConfigurationWr.a_tyDSParam[3].sDownstreamInterfaceId  	:= p_tyRmtSetConfiguration.tyData.a_tyDownstreamConfigurations[p_udiRmtIndexDS4].sDownstreamInterfaceId;
		END_IF

		IF p_tyRmtSetConfiguration.tyAvl.bMachineId = TRUE THEN

			tyConfigurationWr.a_tyUSParam[0].sMachineId		:= p_tyRmtSetConfiguration.tyData.sMachineId;
			tyConfigurationWr.a_tyDSParam[0].sMachineId		:= p_tyRmtSetConfiguration.tyData.sMachineId;
			tyConfigurationWr.tySvyParam.sMachineId		    := p_tyRmtSetConfiguration.tyData.sMachineId;

		END_IF

		IF p_tyRmtSetConfiguration.tyAvl.bSupervisorySystemPort = TRUE THEN

			tyConfigurationWr.tySvyParam.uiSvySvstemPort	:= p_tyRmtSetConfiguration.tyData.uiSupervisorySystemPort;

		END_IF

	ELSIF p_bUISaveHMIConfigure THEN //Save US, DS Configure in HMI

		tyConfigurationWr.a_tyUSParam[0]  := pa_tyUSParam[0]; //lane 1 US
		tyConfigurationWr.a_tyDSParam[0]  := pa_tyDSParam[0]; //lane 1 DS
		tyConfigurationWr.a_tyUSParam[1]  := pa_tyUSParam[1]; //lane 2 US
		tyConfigurationWr.a_tyDSParam[1]  := pa_tyDSParam[1]; //lane 2 DS
		tyConfigurationWr.a_tyUSParam[2]  := pa_tyUSParam[2]; //lane 3 US
		tyConfigurationWr.a_tyDSParam[2]  := pa_tyDSParam[2]; //lane 3 DS
		tyConfigurationWr.a_tyUSParam[3]  := pa_tyUSParam[3]; //lane 4 US
		tyConfigurationWr.a_tyDSParam[3]  := pa_tyDSParam[3]; //lane 4 DS

	ELSIF p_bUISaveHMISvyConfig THEN //Save Supervisory Configure in HMI

		tyConfigurationWr.tySvyParam  := p_tySvyParam;

	END_IF

END_ACTION
```

#### Act_Background_Command.st - Do Not Change!!!
```iecst
(** 2019-05-04 **)
ACTION Act_Background_Command:

	//principal echo command

	//fHermesProcessCmd(ADR(a_tyCommandProcessList),ADR(a_tyCommandPause),ADR(a_usiCommandIdx));

	FOR usiIdx  := 0 TO SIZEOF(a_tyCommandProcessList)/SIZEOF(a_tyCommandProcessList[0]) DO
		IF a_tyCommandProcessList[usiIdx].udiCommandParam = 0 OR a_tyCommandProcessList[usiIdx].udiComMode = 0 OR a_tyCommandProcessList[usiIdx].udiInterfaceString = 0 THEN
			EXIT; //exit if address empty
		END_IF
		p_tyHermesCmdParam ACCESS a_tyCommandProcessList[usiIdx].udiCommandParam;
		p_tyHermesCmdPause ACCESS ADR(a_tyCommandPause[usiIdx]);
		p_tyHermesCmdLockConv ACCESS ADR(a_tyCommandLockInputConv[usiIdx]);
		p_tyHermesCmdOvenInfeed ACCESS ADR(a_tyCommandOvenInfeed[usiIdx]);
		p_udiComMode ACCESS a_tyCommandProcessList[usiIdx].udiComMode;
		//------- Process Rcv and BoardCast if not suppported ------//
		IF p_tyHermesCmdParam.usiCommandIdx <> a_usiCommandIdx[usiIdx] AND p_udiComMode =1 THEN //track command idx
			//Checking Processability and feature
			usiPrevCmdIdx := a_usiCommandIdx[usiIdx];

			//--------------Rcv------------//
			IF p_tyHermesCmdPause.bFeatureRequestTo THEN
				fHermesRcvCmdReqToPause(ADR(a_usiCommandIdx[usiIdx]),ADR(p_tyHermesCmdParam),ADR(p_tyHermesCmdPause));
			END_IF

			IF  p_tyHermesCmdPause.bFeatureRequestFrom THEN
				fHermesRcvCmdReqFromPause(ADR(a_usiCommandIdx[usiIdx]),ADR(p_tyHermesCmdParam),ADR(p_tyHermesCmdPause))	;
			END_IF

			IF p_tyHermesCmdLockConv.bFeatureLockConvFrom THEN
				fHermesRcvCmdReqFromLockCov(ADR(a_usiCommandIdx[usiIdx]),ADR(p_tyHermesCmdParam),ADR(p_tyHermesCmdLockConv))	;
			END_IF

			IF p_tyHermesCmdOvenInfeed.bFeatureOvenInfeedFrom THEN
				fHermesRcvCmdReqFromOvenInfeed(ADR(a_usiCommandIdx[usiIdx]),ADR(p_tyHermesCmdParam),ADR(p_tyHermesCmdOvenInfeed));
			END_IF

			//--------------End of Rcv------------//

			//Adding Command to other interface if not able to execute, Polling
			IF a_usiCommandIdx[usiIdx] = usiPrevCmdIdx THEN 	//if not supported, then broadcast
				FOR usiCmpIdx  := 0 TO SIZEOF(a_tyCommandProcessList)/SIZEOF(a_tyCommandProcessList[0]) DO //loop other
					IF a_tyCommandProcessList[usiCmpIdx].udiCommandParam = 0 OR a_tyCommandProcessList[usiCmpIdx].udiComMode = 0 OR a_tyCommandProcessList[usiCmpIdx].udiInterfaceString = 0 THEN
						EXIT; //exit if address empty
					END_IF
					IF usiIdx <> usiCmpIdx  THEN //not self
						p_sInterface ACCESS a_tyCommandProcessList[usiIdx].udiInterfaceString;
						p_sCmpInterface ACCESS a_tyCommandProcessList[usiCmpIdx].udiInterfaceString;
						p_udiComMode ACCESS a_tyCommandProcessList[usiCmpIdx].udiComMode;
						IF p_sInterface <> p_sCmpInterface AND p_udiComMode = 1 THEN //not same interface and is Hermes Communication
							//message dependant, the oven info need to boardcast to UP only
							p_udiHermesCmpCmdParam ACCESS a_tyCommandProcessList[usiCmpIdx].udiCommandParam;
							IF p_tyHermesCmdParam.eCommand = HermesCommandLockInputConveyor OR p_tyHermesCmdParam.eCommand = HermesCommandUnLockInputConveyor THEN
								IF a_tyCommandProcessList[usiCmpIdx].bUSTrueDSFalse THEN // only to US
									fHermesAddOneCmdTyp(ADR(p_udiHermesCmpCmdParam.a_eCommandSndQ),ADR(p_udiHermesCmpCmdParam.udiMsgCmdBffr),p_tyHermesCmdParam.eCommand);
								END_IF
							ELSIF p_tyHermesCmdParam.eCommand =  HermesCommandOvenInfeed THEN
								IF a_tyCommandProcessList[usiCmpIdx].bUSTrueDSFalse = FALSE THEN // only to DS
									fHermesAddOneCmdTyp(ADR(p_udiHermesCmpCmdParam.a_eCommandSndQ),ADR(p_udiHermesCmpCmdParam.udiMsgCmdBffr),p_tyHermesCmdParam.eCommand);
								END_IF
							ELSE //else dont care up or down
								fHermesAddOneCmdTyp(ADR(p_udiHermesCmpCmdParam.a_eCommandSndQ),ADR(p_udiHermesCmpCmdParam.udiMsgCmdBffr),p_tyHermesCmdParam.eCommand);
							END_IF
						END_IF
					END_IF
				END_FOR
				a_usiCommandIdx[usiIdx] := a_usiCommandIdx[usiIdx] + 1;
			END_IF
		END_IF

		//------- Process Send if supported  ------//
		IF p_tyHermesCmdPause.bFeatureRequestTo THEN
			fHermesSndCmdReqToPause(ADR(p_tyHermesCmdParam),ADR(p_tyHermesCmdPause));
		END_IF

		IF  p_tyHermesCmdPause.bFeatureRequestFrom THEN
			fHermesSndCmdReqFromPause(ADR(p_tyHermesCmdParam),ADR(p_tyHermesCmdPause));
		END_IF

		IF p_tyHermesCmdLockConv.bFeatureLockConvTo THEN
			fHermesSndCmdReqToLockConv(ADR(p_tyHermesCmdParam),ADR(p_tyHermesCmdLockConv));
		END_IF

		IF p_tyHermesCmdOvenInfeed.bFeatureOvenInfeedTo THEN
			fHermesSndCmdReqToOvenInfeed(ADR(p_tyHermesCmdParam),ADR(p_tyHermesCmdOvenInfeed));
		END_IF

	END_FOR

END_ACTION
```

#### Act_Background_Route.st - Do Not Change!!!
```iecst
(** 2021-08-01 **)
ACTION Act_Background_Route:
	//Routing function
	//reverse route, input receiving
	IF NOT(bSwitchtoReverseTransport) THEN
		p_tyUSHermestyBoardAvailable ACCESS p_USHermestyBoardAvailable;
		p_tyDSHermesCurrBASnd ACCESS p_DSHermesBrdAvlSnd;
		p_tyUSRevHermesBFRcv  ACCESS p_USHermes2BrdForecast;
		p_bUSHermesBrdAvlRcved ACCESS p_USHermesBoardAvailableRcved;
		p_bUSRevHermesBrdForecastRcv ACCESS p_USHermes2BrdForecastRcv;
		p_bUSHermesStopTransport ACCESS p_USHermesStopTransportSent;
		p_tyUSHermesStopTransport ACCESS p_USHermesStopTransportSentMsg;
		p_bReceiveReverseUSMcRdy ACCESS p_DSHermesUSRdy;
		pa_tyLinkXMLTableDataBrdAvl ACCESS p_USHermesTableDataBrdAvl;
		p_iLinkXMLTableDataBrdAvlTtlIdx ACCESS p_USHermesTableDataBrdAvlTtlIdx;

		p_bUSCurrHermesBrdForecastRcv ACCESS p_USHermesBrdForecastRcv;
		p_tyUSCurrHermesBFRcv ACCESS p_USHermesBrdForecast;

		p_bDSHermesTransportFinished ACCESS p_DSHermesTransportFinish ;
		p_tyDSHermesTransportFinished ACCESS p_DSHermesTransportFinishMsg;

		p_usiReverseDSSndBfWBrdID ACCESS ADR(usiReverseDS2SndBfWBrdID);
	ELSIF bSwitchtoReverseTransport THEN
		p_tyUSHermestyBoardAvailable ACCESS p_USHermes2tyBoardAvailable;
		p_tyDSHermesCurrBASnd ACCESS p_DSHermes2BrdAvlSnd;
		p_tyUSRevHermesBFRcv  ACCESS p_USHermesBrdForecast;
		p_bUSHermesBrdAvlRcved ACCESS p_USHermes2BoardAvailableRcved;
		p_bUSRevHermesBrdForecastRcv ACCESS  p_USHermesBrdForecastRcv;
		p_bUSHermesStopTransport ACCESS p_USHermes2StopTransportSent;
		p_tyUSHermesStopTransport ACCESS p_USHermes2StopTransportSentMsg;
		p_bReceiveReverseUSMcRdy ACCESS p_DSHermes2USRdy;
		pa_tyLinkXMLTableDataBrdAvl ACCESS p_USHermes2TableDataBrdAvl;
		p_iLinkXMLTableDataBrdAvlTtlIdx ACCESS p_USHermes2TableDataBrdAvlTtlIdx;

		p_bDSHermesTransportFinished ACCESS p_DSHermes2TransportFinish;
		p_tyDSHermesTransportFinished ACCESS p_DSHermes2TransportFinishMsg;

		p_bUSCurrHermesBrdForecastRcv ACCESS p_USHermes2BrdForecastRcv;
		p_tyUSCurrHermesBFRcv ACCESS p_USHermes2BrdForecast;

		p_usiReverseDSSndBfWBrdID ACCESS ADR(usiReverseDS1SndBfWBrdID);
	END_IF
	usiReverseDS1SndBfWBrdID := 0;
	usiReverseDS2SndBfWBrdID := 0;

	IF NOT(p_bReverseReceiveRoute) AND NOT(p_bReverseSentRoute) THEN //flipper on upstream
		bSwitchtoReverseTransport := FALSE;
	ELSE
		IF p_bReverseReceiveRoute THEN //flipper on upstream
			//process Reverse Input
			IF  EDGEPOS(p_bUSRevHermesBrdForecastRcv AND p_tyDSHermesCurrBASnd.tyData.sBoardId = p_tyUSRevHermesBFRcv.tyData.sBoardId AND p_tyUSRevHermesBFRcv.tyData.sBoardId <> '' ) THEN
				//bSwitchtoReverseTransport := NOT(bSwitchtoReverseTransport); //when to reset ReverseRcv back , if the BASnd not the same anymore
				bReqReverseAfterTransptFinished := TRUE;
			ELSIF (EDGEPOS(p_bUSRevHermesBrdForecastRcv AND p_tyUSRevHermesBFRcv.tyData.sBoardId = '' )) THEN
				//OR EDGEPOS(tyMsgTypeRcv.bTransportFinished AND tyTransportFinished.tyData.eTransferState = HermesTransferStateComplete )
				 bReqReverseAfterTransptFinished := FALSE;
			//	bSwitchtoReverseTransport := NOT(bSwitchtoReverseTransport);
			END_IF
			IF bReqReverseAfterTransptFinished AND EDGEPOS(p_bDSHermesTransportFinished AND p_tyDSHermesTransportFinished.tyData.eTransferState  = HermesTransferStateComplete) THEN
				bReqReverseAfterTransptFinished := FALSE;
				bPrevReversalCondition := bSwitchtoReverseTransport;
				bSwitchtoReverseTransport := NOT(bSwitchtoReverseTransport);
			ELSIF bPrevReversalCondition <> bSwitchtoReverseTransport AND EDGEPOS(p_bUSCurrHermesBrdForecastRcv AND p_tyUSCurrHermesBFRcv.tyData.sBoardId = '' ) THEN
				bSwitchtoReverseTransport := bPrevReversalCondition;
			END_IF
		END_IF
		IF p_bReverseSentRoute THEN //flipper on downstream
			//update Reverse Sent
			IF bStopTransportSucceed THEN
				bSelfReverseAfterTransptFinished := TRUE;
			END_IF

			//reset when complete transport or initial run but no board
			IF bBFWithoutBoardID THEN
				bBFWithoutBoardID := FALSE;
				p_usiReverseDSSndBfWBrdID := 2;
			END_IF

			IF bSelfReverseAfterTransptFinished AND  EDGEPOS(p_bDSHermesTransportFinished AND p_tyDSHermesTransportFinished.tyData.eTransferState  = HermesTransferStateComplete) THEN
				bSelfReverseAfterTransptFinished	:= FALSE;
				bSwitchtoReverseTransport := NOT(bSwitchtoReverseTransport);
			ELSIF bSelfReverseAfterTransptFinished AND EDGEPOS(p_bOpsInvertStepInitDone AND NOT(p_bOpsInvertHvBrd)) THEN
				bSelfReverseAfterTransptFinished	:= FALSE;
				bSwitchtoReverseTransport := NOT(bSwitchtoReverseTransport);
				bBFWithoutBoardID := TRUE;
			END_IF

		END_IF
	END_IF

	fbRstReverseRcvGate(IN:= bSwitchtoReverseTransport); //notifty to reset when staying too long in reversal and not board
	bNotifyRstReverseRcvGate := fbRstReverseRcvGate.Q;

	//iGotoLane 0 Default Lane
	//iGotoLane 1 Route1
	//internal condition
	IF NOT(p_bManualRmvRoute OR p_bReturnRoute OR p_bNomRouteEn) THEN
		usiReverseDS1SndBfWBrdID := FALSE;
		usiReverseDS2SndBfWBrdID := FALSE;
		bManualRmvBrdCond := FALSE;
		iGotoLane	:= 0;
		bProcessRouteReversal := FALSE;
		bTriggerRouteReversal := FALSE;
	ELSE
		// intermediate reversal condition
		IF (p_bReturnRoute AND bProcessRouteMachine) AND EDGEPOS(p_bUSHermesBrdAvlRcved AND p_tyUSHermestyBoardAvailable.tyData.iRoute  = 900 ) THEN //flipping station reversal condition
			bProcessRouteReversal := TRUE;
		ELSIF (p_bReturnRoute AND bTriggerRouteMachine) AND EDGEPOS(p_bUSHermesBrdAvlRcved AND p_tyUSHermestyBoardAvailable.tyAvl.bFlippedBoard  AND p_tyUSHermestyBoardAvailable.tyData.eFlippedBoard = HermesFlippedBoardTopSideUp) THEN
			bTriggerRouteReversal := TRUE; //condition link to corresponding inspection zone
		END_IF

		bRouteHaveBeenTriggerred := EDGEPOS(bProcessRouteReversal OR bTriggerRouteReversal);
		bStopTransportFailed := EDGEPOS(p_bUSHermesStopTransport AND (p_tyUSHermesStopTransport.tyData.eTransferState = HermesTransferStateIncomplete OR p_tyUSHermesStopTransport.tyData.eTransferState = HermesTransferStateNotStarted));
		bStopTransportSucceed := EDGEPOS(p_bUSHermesStopTransport AND p_tyUSHermesStopTransport.tyData.eTransferState = HermesTransferStateComplete AND p_bLinkConvHvBrd);

		//receiving Route
		IF	NOT(p_tyUSHermestyBoardAvailable.tyAvl.bRoute)   THEN
			iGotoLane := 0; //default, depend on priority
		ELSE
			IF  p_bManualRmvRoute AND p_tyUSHermestyBoardAvailable.tyData.iRoute  = 999  THEN
				bManualRmvBrdCond := TRUE;

			ELSIF p_bReturnRoute AND (bProcessRouteReversal OR bTriggerRouteReversal)THEN //OR p_usiReverseDSSndBfWBrdID) THEN
				//Reset
				//fbRstReverseDSSndBF(IN:= p_usiReverseDSSndBfWBrdID AND NOT(p_bReceiveReverseUSMcRdy));
				IF bRouteHaveBeenTriggerred THEN
					p_usiReverseDSSndBfWBrdID := 1;
//				ELSIF (p_usiReverseDSSndBfWBrdID AND p_bReceiveReverseUSMcRdy) OR fbRstReverseDSSndBF.Q THEN
//					p_usiReverseDSSndBfWBrdID := 0;
				END_IF

				IF bProcessRouteReversal OR bTriggerRouteReversal  THEN //Route Guide (900),flipper as downstream
					IF bStopTransportFailed THEN
						bProcessRouteReversal := FALSE;
						bTriggerRouteReversal := FALSE;
					ELSIF bStopTransportSucceed  THEN //successful transport
						bSwitchtoReverseTransport := NOT(bSwitchtoReverseTransport);
						FOR i := 0 TO 200 DO
							IF (a_tyHermesBrdAvlData[1].a_tyXMLTableDataBrdAvl[i].sTitle = 'AT') THEN
								fConvertToLower_254(ADR(sLowerCase) , a_tyHermesBrdAvlData[1].a_tyXMLTableDataBrdAvl[i].sValue);
								IF (sLowerCase = 'route') THEN
									IF a_tyHermesBrdAvlData[1].a_tyXMLTableDataBrdAvl[i+1].sTitle = 'AV' THEN
										IF p_tyUSHermestyBoardAvailable.tyData.iRoute = 900 AND bProcessRouteReversal THEN
											a_tyHermesBrdAvlData[1].a_tyXMLTableDataBrdAvl[i+1].sValue	:= '0';
										ELSIF p_tyUSHermestyBoardAvailable.tyData.iRoute <> 900 AND bTriggerRouteReversal  THEN
											a_tyHermesBrdAvlData[1].a_tyXMLTableDataBrdAvl[i+1].sValue	:= '990';
										END_IF
										EXIT;
									END_IF
								END_IF
							END_IF
						END_FOR
						bProcessRouteReversal := FALSE;
						bTriggerRouteReversal := FALSE;
					END_IF
				END_IF

			ELSIF p_bNomRouteEn THEN
				iMinDis := 0;
				FOR usidx := 0 TO 2 DO
					//bChecking Closest Route
					IF p_tyUSHermestyBoardAvailable.tyData.iRoute = tyCurrConfiguration.a_tyDSParam[usidx].iLaneID THEN
						iGotoLane := usidx; //iGotoLane switch direction
						EXIT;
					ELSIF iMinDis = 0 THEN
						iMinDis := ABS(p_tyUSHermestyBoardAvailable.tyData.iRoute - tyCurrConfiguration.a_tyDSParam[usidx].iLaneID);
						iGotoLane := usidx;
					ELSE
						IF iMinDis > ABS(p_tyUSHermestyBoardAvailable.tyData.iRoute - tyCurrConfiguration.a_tyDSParam[usidx].iLaneID) THEN
							iGotoLane := usidx;
							iMinDis := ABS(p_tyUSHermestyBoardAvailable.tyData.iRoute - tyCurrConfiguration.a_tyDSParam[usidx].iLaneID);
						END_IF
					END_IF
				END_FOR
			END_IF

			bEntToReversePosition := bProcessRouteReversal OR bTriggerRouteReversal;
		END_IF

		//Process 900
		//when to reset block DS signal

		//Process 999
		//fbRstReverseDSSndBF(IN:= bManualRmvBrdCond);

	//	bBlkUS := bBlkUS OR bReverseDSSndBfWBrdID; //OR p_bSwitchtoReverseTransport;
	END_IF

END_ACTION
```

#### Act_Alarm.st - Do Not Change!!!
```iecst
(** 2021-08-01 **)
ACTION Act_Alarm:

	//Error
	IF EDGEPOS(eStatus = Error) THEN

		tyAlmData.sProgNm		:= p_sProgNm;
		tyAlmData.udiCode		:= udiStatus;
		tyAlmData.eSeverity		:= AlmSeverityError;
		tyAlmData.udiRunTime	:= tyAlmData.udiRunTime + 1;
		tyAlmData.bAlm			:= TRUE;
		tyAlmData.udiModuleNum  := udiModuleNum;
		g_sHermesProgNm		:= p_sProgNm;

		//Get Error Message
		IF tyAlmData.udiCode < 10000 OR tyAlmData.udiCode > 10099 THEN
			tyAlmData.sAlmMsg	:= 'Unknown';
			tyAlmData.sRcyMsg	:= 'Unknown';
		ELSE
			tyAlmData.sAlmMsg	:= a_tyAlmText[tyAlmData.udiCode].sAlmText;
			tyAlmData.sRcyMsg	:= a_tyAlmText[tyAlmData.udiCode].sRcyText;
		END_IF

		sStatTxt	:= tyAlmData.sAlmMsg;

	ELSIF bRstErr AND (tyAlmData.udiCode <> 0) THEN

		tyAlmData.udiCode	:= 0;
		tyAlmData.eSeverity	:= AlmSeverityNA;
		tyAlmData.sAlmMsg	:= '';
		tyAlmData.sRcyMsg	:= '';
		tyAlmData.bAlm		:= FALSE;

		sStatTxt	:= a_sStatText[eStat];

	END_IF

END_ACTION
```

#### InputRef.var - Do Not Change!!!
```iecst
(*2021-08-01*)
(**)
(*General*)
VAR
	p_eAct : REFERENCE TO eHermesAction;
	p_udiRstErr : REFERENCE TO UDINT;
	p_bPrep : REFERENCE TO BOOL;
	p_bEn : REFERENCE TO BOOL;
	p_bDis : REFERENCE TO BOOL;
END_VAR
(**)
(*Configuration*)
(**)
(*Input*)
VAR
	pa_tyUSParam : REFERENCE TO ARRAY[0..c_diHermesConfigMaxIdx] OF tyHermesUSParam;
	pa_tyDSParam : REFERENCE TO ARRAY[0..c_diHermesConfigMaxIdx] OF tyHermesDSParam;
	p_bRmtPrep : REFERENCE TO BOOL;
	p_bRmtEn : REFERENCE TO BOOL;
	p_tyRmtParam : REFERENCE TO tyHermesRmtParam;
	p_tySvyParam : REFERENCE TO tyHermesSvyParam;
	p_sMcId : REFERENCE TO STRING[30];
	p_bRmtHermesWriteConfig : REFERENCE TO BOOL;
	p_bSvyHermesWriteConfig : REFERENCE TO BOOL;
	p_bUISaveHMIConfigure : REFERENCE TO BOOL;
	p_bUISaveHMISvyConfig : REFERENCE TO BOOL;
	p_tyRmtSetConfiguration : REFERENCE TO tyHermesCurrentConfiguration;
	p_tySvySetConfiguration : REFERENCE TO tyHermesCurrentConfiguration;
	p_bSvyPrep : REFERENCE TO BOOL;
	p_bSvyEn : REFERENCE TO BOOL;
	p_sRetainFileName1 : REFERENCE TO STRING[80];
	p_sRetainFileName2 : REFERENCE TO STRING[80];
	p_sRetainFileName3 : REFERENCE TO STRING[80];
	p_sRetainFileName4 : REFERENCE TO STRING[80];
	p_udiRetainDataAddr1 : REFERENCE TO UDINT;
	p_udiRetainDataLen1 : REFERENCE TO UDINT;
	p_udiRetainDataAddr2 : REFERENCE TO UDINT;
	p_udiRetainDataLen2 : REFERENCE TO UDINT;
	p_udiRetainDataAddr3 : REFERENCE TO UDINT;
	p_udiRetainDataLen3 : REFERENCE TO UDINT;
	p_udiRetainDataAddr4 : REFERENCE TO UDINT;
	p_udiRetainDataLen4 : REFERENCE TO UDINT;
	p_sConfigFileName : REFERENCE TO STRING[80];
	p_sProgNm : REFERENCE TO STRING[15];
	p_bNtSettingsLoadDone : REFERENCE TO BOOL;
	p_bNTParamUnlockCovPrep : REFERENCE TO BOOL;
	p_bNTParamMachineSafetySig : REFERENCE TO BOOL;
END_VAR
(*Route*)
VAR
	p_tyDSHermesCurrBASnd : REFERENCE TO tyHermesBoardAvailable;
	p_bUSRevHermesBrdForecastRcv : REFERENCE TO BOOL;
	p_tyUSRevHermesBFRcv : REFERENCE TO tyHermesBoardForecast;
	p_bUSCurrHermesBrdForecastRcv : REFERENCE TO BOOL;
	p_tyUSCurrHermesBFRcv : REFERENCE TO tyHermesBoardForecast;
	p_tyUSHermesStopTransport : REFERENCE TO tyHermesStopTransport;
	p_bUSHermesBrdAvlRcved : REFERENCE TO BOOL;
	p_bUSHermesStopTransport : REFERENCE TO BOOL;
	p_bReverseReceiveRoute : REFERENCE TO BOOL;
	p_bReverseSentRoute : REFERENCE TO BOOL;
	p_bManualRmvRoute : REFERENCE TO BOOL;
	p_bReturnRoute : REFERENCE TO BOOL;
	p_bNomRouteEn : REFERENCE TO BOOL;
	p_bReceiveReverseUSMcRdy : REFERENCE TO BOOL;
	p_usiReverseDSSndBfWBrdID : REFERENCE TO USINT;
	p_bDSHermesTransportFinished : REFERENCE TO BOOL;
	p_tyDSHermesTransportFinished : REFERENCE TO tyHermesTransportFinished;
	p_bOpsInvertStepInitDone : REFERENCE TO BOOL;
	p_bOpsInvertHvBrd : REFERENCE TO BOOL;
END_VAR
(*Gate Configuration*)
(*RmtHermes*)
VAR
	p_bRmtFoundIndexUS1 : REFERENCE TO BOOL;
	p_bRmtFoundIndexUS2 : REFERENCE TO BOOL;
	p_bRmtFoundIndexUS3 : REFERENCE TO BOOL;
	p_bRmtFoundIndexUS4 : REFERENCE TO BOOL;
	p_bRmtFoundIndexDS1 : REFERENCE TO BOOL;
	p_bRmtFoundIndexDS2 : REFERENCE TO BOOL;
	p_bRmtFoundIndexDS3 : REFERENCE TO BOOL;
	p_bRmtFoundIndexDS4 : REFERENCE TO BOOL;
	p_udiRmtIndexUS1 : REFERENCE TO UDINT;
	p_udiRmtIndexUS2 : REFERENCE TO UDINT;
	p_udiRmtIndexUS3 : REFERENCE TO UDINT;
	p_udiRmtIndexUS4 : REFERENCE TO UDINT;
	p_udiRmtIndexDS1 : REFERENCE TO UDINT;
	p_udiRmtIndexDS2 : REFERENCE TO UDINT;
	p_udiRmtIndexDS3 : REFERENCE TO UDINT;
	p_udiRmtIndexDS4 : REFERENCE TO UDINT;
END_VAR
(**)
(*SvyHermes*)
VAR
	p_bSvyFoundIndexUS1 : REFERENCE TO BOOL;
	p_bSvyFoundIndexUS2 : REFERENCE TO BOOL;
	p_bSvyFoundIndexUS3 : REFERENCE TO BOOL;
	p_bSvyFoundIndexUS4 : REFERENCE TO BOOL;
	p_bSvyFoundIndexDS1 : REFERENCE TO BOOL;
	p_bSvyFoundIndexDS2 : REFERENCE TO BOOL;
	p_bSvyFoundIndexDS3 : REFERENCE TO BOOL;
	p_bSvyFoundIndexDS4 : REFERENCE TO BOOL;
	p_udiSvyIndexUS1 : REFERENCE TO UDINT;
	p_udiSvyIndexUS2 : REFERENCE TO UDINT;
	p_udiSvyIndexUS3 : REFERENCE TO UDINT;
	p_udiSvyIndexUS4 : REFERENCE TO UDINT;
	p_udiSvyIndexDS1 : REFERENCE TO UDINT;
	p_udiSvyIndexDS2 : REFERENCE TO UDINT;
	p_udiSvyIndexDS3 : REFERENCE TO UDINT;
	p_udiSvyIndexDS4 : REFERENCE TO UDINT;
END_VAR
(**)
(*Local Pointer for Cmd*)
VAR
	p_tyHermesCmdParam : REFERENCE TO tyHermesCommandParam;
	p_udiHermesCmpCmdParam : REFERENCE TO tyHermesCommandParam;
	p_tyHermesCmdPause : REFERENCE TO tyHermesCommandPause;
	p_tyHermesCmdLockConv : REFERENCE TO tyHermesCommandLockConv;
	p_tyHermesCmdOvenInfeed : REFERENCE TO tyHermesCommandOvenInfeed;
	p_sCmpInterface : REFERENCE TO STRING[80];
	p_sInterface : REFERENCE TO STRING[80];
	p_udiComMode : REFERENCE TO UDINT;
END_VAR
```

#### Local.var - Do Not Change!!!
```iecst
(*2021-08-01*)
(**)
(*Local Action, State & Status*)
VAR
	eAct : eHermesAction := HermesActIdle;
	eStat : eHermesAction := HermesActIdle;
	eStatus : eFBStatus := Idle;
	udiStatus : UDINT := 0;
	sStatTxt : STRING[200] := '';
	a_sStatText : ARRAY[0..50] OF STRING[200] := ['Idling','Background Starting Operations','Background Stopping Operations','Deleting Old Log File','Creating Directory','Writing Retain File','Reading Retain File','Writing Configuration File','Reading Configuration File',42('')];
END_VAR
(**)
(*Local Alarm*)
VAR
	tyAlmData : tyAlmDat;
	a_tyAlmText : ARRAY[10000..10099] OF tyAlmTxt := [(sAlmText:='Create User Directory Error',sRcyText:='An Error Occurred While Attempting To Create User Directory. Please Contact Nutek For A Possible Solution'),(sAlmText:='Create Retain Directory Error',sRcyText:='An Error Occurred While Attempting To Create Retain Directory. Please Contact Nutek For A Possible Solution'),(sAlmText:='File Open Error While Reading Retain File',sRcyText:='An Error Was Encountered While Trying To Open File. Please Contact Nutek For A Possible Solution.'),(sAlmText:='File Read Error While Reading Retain File',sRcyText:='An Error Was Encountered While Trying To Read File. Please Contact Nutek For A Possible Solution.'),(sAlmText:='File Close Error While Reading Retain File',sRcyText:='An Error Was Encountered While Trying To Close File. Please Contact Nutek For A Possible Solution.'),(sAlmText:='File Open Error While Writing Retain File',sRcyText:='An Error Was Encountered While Trying To Open File. Please Contact Nutek For A Possible Solution.'),(sAlmText:='File Create Error While Writing Retain File',sRcyText:='An Error Was Encountered While Trying To Create File. Please Contact Nutek For A Possible Solution.'),(sAlmText:='File Write Error While Writing Retain File',sRcyText:='An Error Was Encountered While Trying To Write File. Please Contact Nutek For A Possible Solution.'),(sAlmText:='File Close Error While Writing Retain File',sRcyText:='An Error Was Encountered While Trying To Close File. Please Contact Nutek For A Possible Solution.'),(sAlmText:='Directory Does Not Exist While Writing Retain File',sRcyText:='The Directory Does Not Exist. Please Contact Nutek For A Possible Solution.'),(sAlmText:='Create Log Directory Error',sRcyText:='An Error Occurred While Attempting To Create Log Directory. Please Contact Nutek For A Possible Solution'),(sAlmText:='Create Machine Parameter Directory Error',sRcyText:='An Error Occurred While Attempting To Create Machine Parameter Directory. Please Contact Nutek For A Possible Solution'),(sAlmText:='File Open Error While Reading Config File',sRcyText:='An Error Was Encountered While Trying To Open File. Please Contact Nutek For A Possible Solution.'),(sAlmText:='File Read Error While Reading Config File',sRcyText:='An Error Was Encountered While Trying To Read File. Please Contact Nutek For A Possible Solution.'),(sAlmText:='File Close Error While Reading Config File',sRcyText:='An Error Was Encountered While Trying To Close File. Please Contact Nutek For A Possible Solution.'),(sAlmText:='File Open Error While Writing Config File',sRcyText:='An Error Was Encountered While Trying To Open File. Please Contact Nutek For A Possible Solution.'),(sAlmText:='File Create Error While Writing Config File',sRcyText:='An Error Was Encountered While Trying To Create File. Please Contact Nutek For A Possible Solution.'),(sAlmText:='File Write Error While Writing Config File',sRcyText:='An Error Was Encountered While Trying To Write File. Please Contact Nutek For A Possible Solution.'),(sAlmText:='File Close Error While Writing Config File',sRcyText:='An Error Was Encountered While Trying To Close File. Please Contact Nutek For A Possible Solution.'),(sAlmText:='Directory Does Not Exist While Writing Config File',sRcyText:='The Directory Does Not Exist. Please Contact Nutek For A Possible Solution.'),(0),2(0),3((0)),0,3((0)),(sAlmText:='File Open Error While Writing Retain File Lane 2',sRcyText:='An Error Was Encountered While Trying To Open File. Please Contact Nutek For A Possible Solution.'),(0),(sAlmText:='File Open Error While Reading Lane 2 Retain File',sRcyText:='An Error Was Encountered While Trying To Open File. Please Contact Nutek For A Possible Solution.'),(sAlmText:='File Read Error While Reading Lane 2 Retain File',sRcyText:='An Error Was Encountered While Trying To Read File. Please Contact Nutek For A Possible Solution.'),(sAlmText:='File Close Error While Reading Lane 2 Retain File',sRcyText:='An Error Was Encountered While Trying To Close File. Please Contact Nutek For A Possible Solution.'),(sAlmText:='File Open Error While Writing Lane 2 Retain File',sRcyText:='An Error Was Encountered While Trying To Open File. Please Contact Nutek For A Possible Solution.'),(sAlmText:='File Create Error While Writing Lane 2 Retain File',sRcyText:='An Error Was Encountered While Trying To Create File. Please Contact Nutek For A Possible Solution.'),(sAlmText:='File Write Error While Writing Lane 2 Retain File',sRcyText:='An Error Was Encountered While Trying To Write File. Please Contact Nutek For A Possible Solution.'),(sAlmText:='File Close Error While Writing Lane 2 Retain File',sRcyText:='An Error Was Encountered While Trying To Close File. Please Contact Nutek For A Possible Solution.'),(sAlmText:='Directory Does Not Exist While Writing Lane 2 Retain File',sRcyText:='The Directory Does Not Exist. Please Contact Nutek For A Possible Solution.'),2((0)),(sAlmText:='File Open Error While Reading Lane 3 Retain File',sRcyText:='An Error Was Encountered While Trying To Open File. Please Contact Nutek For A Possible Solution.'),(sAlmText:='File Read Error While Reading Lane 3 Retain File',sRcyText:='An Error Was Encountered While Trying To Read File. Please Contact Nutek For A Possible Solution.'),(sAlmText:='File Close Error While Reading Lane 3 Retain File',sRcyText:='An Error Was Encountered While Trying To Close File. Please Contact Nutek For A Possible Solution.'),(sAlmText:='File Open Error While Writing Lane 3 Retain File',sRcyText:='An Error Was Encountered While Trying To Open File. Please Contact Nutek For A Possible Solution.'),(sAlmText:='File Create Error While Writing Lane 3 Retain File',sRcyText:='An Error Was Encountered While Trying To Create File. Please Contact Nutek For A Possible Solution.'),(sAlmText:='File Write Error While Writing Lane 3 Retain File',sRcyText:='An Error Was Encountered While Trying To Write File. Please Contact Nutek For A Possible Solution.'),(sAlmText:='File Close Error While Writing Lane 3 Retain File',sRcyText:='An Error Was Encountered While Trying To Close File. Please Contact Nutek For A Possible Solution.'),(sAlmText:='Directory Does Not Exist While Writing Lane 3 Retain File',sRcyText:='The Directory Does Not Exist. Please Contact Nutek For A Possible Solution.'),2((0)),(sAlmText:='File Open Error While Reading Lane 4 Retain File',sRcyText:='An Error Was Encountered While Trying To Open File. Please Contact Nutek For A Possible Solution.'),(sAlmText:='File Read Error While Reading Lane 4 Retain File',sRcyText:='An Error Was Encountered While Trying To Read File. Please Contact Nutek For A Possible Solution.'),(sAlmText:='File Close Error While Reading Lane 4 Retain File',sRcyText:='An Error Was Encountered While Trying To Close File. Please Contact Nutek For A Possible Solution.'),(sAlmText:='File Open Error While Writing Lane 4 Retain File',sRcyText:='An Error Was Encountered While Trying To Open File. Please Contact Nutek For A Possible Solution.'),(sAlmText:='File Create Error While Writing Lane 4 Retain File',sRcyText:='An Error Was Encountered While Trying To Create File. Please Contact Nutek For A Possible Solution.'),(sAlmText:='File Write Error While Writing Lane 4 Retain File',sRcyText:='An Error Was Encountered While Trying To Write File. Please Contact Nutek For A Possible Solution.'),(sAlmText:='File Close Error While Writing Lane 4 Retain File',sRcyText:='An Error Was Encountered While Trying To Close File. Please Contact Nutek For A Possible Solution.'),(sAlmText:='Directory Does Not Exist While Writing Lane 4 Retain File',sRcyText:='The Directory Does Not Exist. Please Contact Nutek For A Possible Solution.'),40((0))];
END_VAR
(**)
(*Local Output*)
VAR
	bFileNotFound : BOOL;
	tyConfiguration : tyHermesConfiguration;
	tyCurrConfiguration : tyHermesConfiguration;
	tyConfigurationWr : tyHermesConfiguration;
END_VAR
(**)
(*Local Input*)
VAR
	udiRstErr : UDINT := 0;
	bPrep : BOOL := TRUE;
	bEn : BOOL := TRUE;
	bDis : BOOL := FALSE;
	a_tyUSParam : ARRAY[0..c_diHermesConfigMaxIdx] OF tyHermesUSParam;
	a_tyDSParam : ARRAY[0..c_diHermesConfigMaxIdx] OF tyHermesDSParam;
	bRmtPrep : BOOL := FALSE;
	bRmtEn : BOOL := FALSE;
	sRetainFileName : STRING[80] := 'Hermes.dat';
	udiRetainDataAddr : UDINT;
	udiRetainDataLen : UDINT;
	tyRmtParam : tyHermesRmtParam;
	tySvyParam : tyHermesSvyParam;
	tyRmtSetConfiguration : tyHermesCurrentConfiguration;
	tySvySetConfiguration : tyHermesCurrentConfiguration;
	bSvyPrep : BOOL := FALSE;
	bSvyEn : BOOL := FALSE;
	sRetainFileName1 : STRING[80] := 'HermesLane1.dat';
	sRetainFileName2 : STRING[80] := 'HermesLane2.dat';
	sRetainFileName3 : STRING[80] := 'HermesLane3.dat';
	sRetainFileName4 : STRING[80] := 'HermesLane4.dat';
	udiRetainDataAddr1 : UDINT;
	udiRetainDataLen1 : UDINT;
	udiRetainDataAddr2 : UDINT;
	udiRetainDataLen2 : UDINT;
	udiRetainDataAddr3 : UDINT;
	udiRetainDataLen3 : UDINT;
	udiRetainDataAddr4 : UDINT;
	udiRetainDataLen4 : UDINT;
	sConfigFileName : STRING[80] := 'Hermes.dat';
	sProgNm : STRING[15] := 'Hermes';
	bNtSettingsLoadDone : BOOL := TRUE;
	bRmtHermesWriteConfig : BOOL := TRUE;
	bSvyHermesWriteConfig : BOOL := TRUE;
	bUISaveHMIConfigure : BOOL := TRUE;
	bUISaveHMISvyConfig : BOOL := TRUE;
	sMcId : STRING[30] := '';
	bRmtFoundIndexUS1 : BOOL := FALSE;
	bRmtFoundIndexUS2 : BOOL := FALSE;
	bRmtFoundIndexUS3 : BOOL := FALSE;
	bRmtFoundIndexUS4 : BOOL := FALSE;
	bRmtFoundIndexDS1 : BOOL := FALSE;
	bRmtFoundIndexDS2 : BOOL := FALSE;
	bRmtFoundIndexDS3 : BOOL := FALSE;
	bRmtFoundIndexDS4 : BOOL := FALSE;
	udiRmtIndexUS1 : UDINT := 0;
	udiRmtIndexUS2 : UDINT := 0;
	udiRmtIndexUS3 : UDINT := 0;
	udiRmtIndexUS4 : UDINT := 0;
	udiRmtIndexDS1 : UDINT := 0;
	udiRmtIndexDS2 : UDINT := 0;
	udiRmtIndexDS3 : UDINT := 0;
	udiRmtIndexDS4 : UDINT := 0;
	bSvyFoundIndexUS1 : BOOL := FALSE;
	bSvyFoundIndexUS2 : BOOL := FALSE;
	bSvyFoundIndexUS3 : BOOL := FALSE;
	bSvyFoundIndexUS4 : BOOL := FALSE;
	bSvyFoundIndexDS1 : BOOL := FALSE;
	bSvyFoundIndexDS2 : BOOL := FALSE;
	bSvyFoundIndexDS3 : BOOL := FALSE;
	bSvyFoundIndexDS4 : BOOL := FALSE;
	udiSvyIndexUS1 : UDINT := 0;
	udiSvyIndexUS2 : UDINT := 0;
	udiSvyIndexUS3 : UDINT := 0;
	udiSvyIndexUS4 : UDINT := 0;
	udiSvyIndexDS1 : UDINT := 0;
	udiSvyIndexDS2 : UDINT := 0;
	udiSvyIndexDS3 : UDINT := 0;
	udiSvyIndexDS4 : UDINT := 0;
END_VAR
(**)
(*Local*)
VAR
	bRstErr : BOOL;
	udiRstErrOld : UDINT;
	bInitDone : BOOL;
	bInitialDone : BOOL;
	bHermesWriteRetainLane1 : BOOL;
	bHermesWriteRetainLane2 : BOOL;
	bHermesWriteRetainLane3 : BOOL;
	bHermesWriteRetainLane4 : BOOL;
	usiStep : USINT;
	tyConfigurationLocal : tyHermesConfiguration;
	tyConfigurationHMI : tyHermesConfiguration;
	eStatOld : eHermesAction := HermesActIdle;
	fbDirCreate1 : fbDirCreate;
	fbDirCreate2 : fbDirCreate;
	fbDirCreate3 : fbDirCreate;
	fbDirCreate4 : fbDirCreate;
	fbFileRead1 : fbFileFullRead;
	fbFileWrite1 : fbFileFullWrite;
	fbFileRead2 : fbFileFullRead;
	fbFileWrite2 : fbFileFullWrite;
	fbFileRead3 : fbFileFullRead;
	fbFileWrite3 : fbFileFullWrite;
	fbFileRead4 : fbFileFullRead;
	fbFileWrite4 : fbFileFullWrite;
	fbFileRead5 : fbFileFullRead;
	fbFileWrite5 : fbFileFullWrite;
	i : INT;
	usiUSHermesCommand : USINT;
	usiDSHermesCommand : USINT;
	usiProcessCmdBffr : USINT;
	a_tyCommandProcessList : ARRAY[0..c_diHermesConfigMaxInterfaceIdx] OF tyHermesCmdProcessList;
	a_tyCommandPause : ARRAY[0..c_diHermesConfigMaxInterfaceIdx] OF tyHermesCommandPause;
	a_tyCommandLockInputConv : ARRAY[0..c_diHermesConfigMaxInterfaceIdx] OF tyHermesCommandLockConv;
	a_tyCommandOvenInfeed : ARRAY[0..c_diHermesConfigMaxInterfaceIdx] OF tyHermesCommandOvenInfeed;
	a_usiCommandIdx : ARRAY[0..c_diHermesConfigMaxInterfaceIdx] OF USINT;
	usiIdx : USINT;
	usiCmpIdx : USINT;
	usiPrevCmdIdx : USINT;
	usiDSIdent : USINT;
	usiUSIdent : USINT;
	usiUSIdent2 : USINT;
	bCmdInitialCompl : BOOL;
	udiModuleNum : UDINT := 2901;
END_VAR
(*route*)
VAR
	bBFWithoutBoardID : BOOL;
	bSwitchtoReverseTransport : BOOL;
	bReqReverseAfterTransptFinished : BOOL;
	bSelfReverseAfterTransptFinished : BOOL;
	bPrevReversalCondition : BOOL;
	bNotifyRstReverseRcvGate : BOOL;
	bReverseReceiveRoute : BOOL;
	bReverseSendRoute : BOOL;
	bProcessRouteMachine : BOOL;
	bTriggerRouteMachine : BOOL;
	bProcessRouteReversal : BOOL;
	bEntToReversePosition : USINT;
	bTriggerRouteReversal : BOOL;
	bRouteHaveBeenTriggerred : BOOL;
	bStopTransportSucceed : BOOL;
	bStopTransportFailed : BOOL;
	iGotoLane : INT;
	fbRstReverseRcvGate : TON;
	fbRstReverseDSSndBF : TON := (PT:=T#2m);
	bManualRmvBrdCond : BOOL;
	usidx : USINT;
	iMinDis : INT;
	bManualRmvRoute : BOOL;
	bReturnRoute : BOOL;
	bNomRouteEn : BOOL;
	usiReverseDS1SndBfWBrdID : USINT;
	usiReverseDS2SndBfWBrdID : USINT;
END_VAR
```
